    |   movel([0.327897, -1.235009, -2.660401, -0.816979, 1.570796, 1.898693],accel_mss,speed_ms,0,blend_radius_m)
    |   movel([0.327586, -1.234473, -2.660677, -0.817239, 1.570796, 1.898382],accel_mss,speed_ms,0,blend_radius_m)
    |   speed_ms = 0.005
    |   movel([0.327586, -1.224931, -2.656020, -0.831439, 1.570796, 1.898382],accel_mss,speed_ms,0,blend_radius_m)
    |   speed_ms = 0.040
    |   movel([0.337842, -1.232613, -2.652083, -0.827693, 1.570796, 1.908639],accel_mss,speed_ms,0,blend_radius_m)
    |   speed_ms = 0.005
    |   movel([0.337842, -1.242122, -2.656705, -0.813562, 1.570796, 1.908639],accel_mss,speed_ms,0,blend_radius_m)
    |   speed_ms = 0.025
    |   movel([0.336390, -1.242228, -2.656649, -0.813511, 1.570796, 1.907187],accel_mss,speed_ms,0,blend_radius_m)
    |   movel([0.335495, -1.242155, -2.656688, -0.813546, 1.570796, 1.906292],accel_mss,speed_ms,0,blend_radius_m)
    |   movel([0.333990, -1.241944, -2.656798, -0.813647, 1.570796, 1.904786],accel_mss,speed_ms,0,blend_radius_m)
    |   movel([0.333947, -1.242489, -2.656513, -0.813387, 1.570796, 1.904743],accel_mss,speed_ms,0,blend_radius_m)
    |   movel([0.333924, -1.243378, -2.656047, -0.812965, 1.570796, 1.904720],accel_mss,speed_ms,0,blend_radius_m)
    |   movel([0.333526, -1.244120, -2.655656, -0.812612, 1.570796, 1.904322],accel_mss,speed_ms,0,blend_radius_m)
    |   movel([0.333176, -1.244437, -2.655490, -0.812462, 1.570796, 1.903972],accel_mss,speed_ms,0,blend_radius_m)
    |   movel([0.332782, -1.244663, -2.655370, -0.812355, 1.570796, 1.903579],accel_mss,speed_ms,0,blend_radius_m)
    |   movel([0.331750, -1.244958, -2.655215, -0.812216, 1.570796, 1.902546],accel_mss,speed_ms,0,blend_radius_m)
    |   movel([0.330907, -1.245181, -2.655098, -0.812111, 1.570796, 1.901703],accel_mss,speed_ms,0,blend_radius_m)
    |   movel([0.331284, -1.245824, -2.654758, -0.811807, 1.570796, 1.902081],accel_mss,speed_ms,0,blend_radius_m)
    |   movel([0.331806, -1.246356, -2.654477, -0.811556, 1.570796, 1.902602],accel_mss,speed_ms,0,blend_radius_m)
    |   movel([0.333454, -1.247963, -2.653625, -0.810800, 1.570796, 1.904250],accel_mss,speed_ms,0,blend_radius_m)
    |   movel([0.333871, -1.248606, -2.653284, -0.810499, 1.570796, 1.904667],accel_mss,speed_ms,0,blend_radius_m)
    |   movel([0.333836, -1.249059, -2.653043, -0.810286, 1.570796, 1.904633],accel_mss,speed_ms,0,blend_radius_m)
    |   movel([0.333484, -1.249416, -2.652853, -0.810120, 1.570796, 1.904280],accel_mss,speed_ms,0,blend_radius_m)
    |   movel([0.333131, -1.249421, -2.652851, -0.810117, 1.570796, 1.903927],accel_mss,speed_ms,0,blend_radius_m)
    |   movel([0.332061, -1.248584, -2.653296, -0.810509, 1.570796, 1.902858],accel_mss,speed_ms,0,blend_radius_m)
    |   movel([0.329590, -1.246252, -2.654532, -0.811605, 1.570796, 1.900386],accel_mss,speed_ms,0,blend_radius_m)
    |   movel([0.329051, -1.245580, -2.654887, -0.811922, 1.570796, 1.899848],accel_mss,speed_ms,0,blend_radius_m)
    |   movel([0.328887, -1.245037, -2.655174, -0.812179, 1.570796, 1.899684],accel_mss,speed_ms,0,blend_radius_m)
    |   movel([0.329075, -1.244647, -2.655379, -0.812363, 1.570796, 1.899871],accel_mss,speed_ms,0,blend_radius_m)
    |   movel([0.329758, -1.244331, -2.655545, -0.812513, 1.570796, 1.900555],accel_mss,speed_ms,0,blend_radius_m)
    |   movel([0.330219, -1.244220, -2.655604, -0.812565, 1.570796, 1.901015],accel_mss,speed_ms,0,blend_radius_m)
    |   movel([0.332711, -1.243637, -2.655910, -0.812842, 1.570796, 1.903507],accel_mss,speed_ms,0,blend_radius_m)
    |   movel([0.332571, -1.242862, -2.656318, -0.813210, 1.570796, 1.903368],accel_mss,speed_ms,0,blend_radius_m)
    |   movel([0.332085, -1.240846, -2.657373, -0.814171, 1.570796, 1.902881],accel_mss,speed_ms,0,blend_radius_m)
    |   movel([0.332184, -1.240399, -2.657606, -0.814384, 1.570796, 1.902980],accel_mss,speed_ms,0,blend_radius_m)
    |   movel([0.332457, -1.240129, -2.657746, -0.814513, 1.570796, 1.903254],accel_mss,speed_ms,0,blend_radius_m)
    |   movel([0.332852, -1.240044, -2.657791, -0.814554, 1.570796, 1.903648],accel_mss,speed_ms,0,blend_radius_m)
    |   movel([0.335457, -1.240841, -2.657375, -0.814173, 1.570796, 1.906254],accel_mss,speed_ms,0,blend_radius_m)
    |   movel([0.336114, -1.240976, -2.657305, -0.814108, 1.570796, 1.906911],accel_mss,speed_ms,0,blend_radius_m)
    |   movel([0.337508, -1.240998, -2.657293, -0.814098, 1.570796, 1.908304],accel_mss,speed_ms,0,blend_radius_m)
    |   movel([0.338667, -1.240917, -2.657336, -0.814137, 1.570796, 1.909464],accel_mss,speed_ms,0,blend_radius_m)
    |   movel([0.339093, -1.240957, -2.657315, -0.814118, 1.570796, 1.909889],accel_mss,speed_ms,0,blend_radius_m)
    |   movel([0.339216, -1.241123, -2.657228, -0.814038, 1.570796, 1.910012],accel_mss,speed_ms,0,blend_radius_m)
    |   movel([0.338972, -1.241703, -2.656925, -0.813761, 1.570796, 1.909768],accel_mss,speed_ms,0,blend_radius_m)
    |   movel([0.338768, -1.241870, -2.656837, -0.813682, 1.570796, 1.909564],accel_mss,speed_ms,0,blend_radius_m)
    |   movel([0.337842, -1.242122, -2.656705, -0.813562, 1.570796, 1.908639],accel_mss,speed_ms,0,blend_radius_m)
    |   movel([0.336390, -1.242228, -2.656649, -0.813511, 1.570796, 1.907187],accel_mss,speed_ms,0,blend_radius_m)
    |   movel([0.335495, -1.242155, -2.656688, -0.813546, 1.570796, 1.906292],accel_mss,speed_ms,0,blend_radius_m)
    |   movel([0.335218, -1.242116, -2.656708, -0.813564, 1.570796, 1.906015],accel_mss,speed_ms,0,blend_radius_m)
    |   speed_ms = 0.005
    |   movel([0.335218, -1.232607, -2.652086, -0.827696, 1.570796, 1.906015],accel_mss,speed_ms,0,blend_radius_m)
    |   speed_ms = 0.040
    |   movel([0.344776, -1.237105, -2.649749, -0.825535, 1.570796, 1.915573],accel_mss,speed_ms,0,blend_radius_m)
    |   speed_ms = 0.005
    |   movel([0.344776, -1.246594, -2.654351, -0.811444, 1.570796, 1.915573],accel_mss,speed_ms,0,blend_radius_m)
    |   speed_ms = 0.025
    |   movel([0.344962, -1.247047, -2.654111, -0.811231, 1.570796, 1.915759],accel_mss,speed_ms,0,blend_radius_m)
    |   movel([0.345103, -1.247442, -2.653902, -0.811045, 1.570796, 1.915899],accel_mss,speed_ms,0,blend_radius_m)
    |   movel([0.345193, -1.247835, -2.653693, -0.810860, 1.570796, 1.915990],accel_mss,speed_ms,0,blend_radius_m)
    |   movel([0.343853, -1.247462, -2.653891, -0.811035, 1.570796, 1.914649],accel_mss,speed_ms,0,blend_radius_m)
    |   movel([0.343381, -1.247399, -2.653925, -0.811065, 1.570796, 1.914177],accel_mss,speed_ms,0,blend_radius_m)
    |   movel([0.342236, -1.247467, -2.653889, -0.811033, 1.570796, 1.913033],accel_mss,speed_ms,0,blend_radius_m)
    |   movel([0.340990, -1.247651, -2.653791, -0.810947, 1.570796, 1.911786],accel_mss,speed_ms,0,blend_radius_m)
    |   movel([0.341964, -1.245315, -2.655027, -0.812047, 1.570796, 1.912761],accel_mss,speed_ms,0,blend_radius_m)
    |   movel([0.342301, -1.244772, -2.655313, -0.812304, 1.570796, 1.913097],accel_mss,speed_ms,0,blend_radius_m)
    |   movel([0.342917, -1.244066, -2.655685, -0.812638, 1.570796, 1.913714],accel_mss,speed_ms,0,blend_radius_m)
    |   movel([0.343093, -1.244020, -2.655709, -0.812660, 1.570796, 1.913889],accel_mss,speed_ms,0,blend_radius_m)
    |   movel([0.343277, -1.244144, -2.655644, -0.812601, 1.570796, 1.914074],accel_mss,speed_ms,0,blend_radius_m)
    |   movel([0.343671, -1.244629, -2.655388, -0.812371, 1.570796, 1.914468],accel_mss,speed_ms,0,blend_radius_m)
    |   movel([0.344776, -1.246594, -2.654351, -0.811444, 1.570796, 1.915573],accel_mss,speed_ms,0,blend_radius_m)
    |   movel([0.344962, -1.247047, -2.654111, -0.811231, 1.570796, 1.915759],accel_mss,speed_ms,0,blend_radius_m)
    |   movel([0.345103, -1.247442, -2.653902, -0.811045, 1.570796, 1.915899],accel_mss,speed_ms,0,blend_radius_m)
    |   movel([0.345193, -1.247835, -2.653693, -0.810860, 1.570796, 1.915990],accel_mss,speed_ms,0,blend_radius_m)
    |   movel([0.344251, -1.247571, -2.653834, -0.810985, 1.570796, 1.915047],accel_mss,speed_ms,0,blend_radius_m)
    |   speed_ms = 0.005
    |   movel([0.344251, -1.238086, -2.649236, -0.825066, 1.570796, 1.915047],accel_mss,speed_ms,0,blend_radius_m)
    |   speed_ms = 0.040
    |   movel([0.347433, -1.243638, -2.646313, -0.822438, 1.570796, 1.918229],accel_mss,speed_ms,0,blend_radius_m)
    |   speed_ms = 0.005
    |   movel([0.347433, -1.253097, -2.650885, -0.808407, 1.570796, 1.918229],accel_mss,speed_ms,0,blend_radius_m)
    |   speed_ms = 0.025
    |   movel([0.347850, -1.253561, -2.650636, -0.808192, 1.570796, 1.918646],accel_mss,speed_ms,0,blend_radius_m)
    |   movel([0.346822, -1.254725, -2.650010, -0.807654, 1.570796, 1.917619],accel_mss,speed_ms,0,blend_radius_m)
    |   movel([0.346418, -1.255196, -2.649756, -0.807437, 1.570796, 1.917215],accel_mss,speed_ms,0,blend_radius_m)
    |   movel([0.345672, -1.256232, -2.649197, -0.806961, 1.570796, 1.916468],accel_mss,speed_ms,0,blend_radius_m)
    |   movel([0.345493, -1.256601, -2.648997, -0.806791, 1.570796, 1.916289],accel_mss,speed_ms,0,blend_radius_m)
    |   movel([0.345323, -1.256697, -2.648945, -0.806747, 1.570796, 1.916119],accel_mss,speed_ms,0,blend_radius_m)
    |   movel([0.345210, -1.256550, -2.649025, -0.806815, 1.570796, 1.916007],accel_mss,speed_ms,0,blend_radius_m)
    |   movel([0.345305, -1.255281, -2.649710, -0.807398, 1.570796, 1.916101],accel_mss,speed_ms,0,blend_radius_m)
    |   movel([0.345190, -1.254371, -2.650200, -0.807817, 1.570796, 1.915986],accel_mss,speed_ms,0,blend_radius_m)
    |   movel([0.344521, -1.252694, -2.651102, -0.808594, 1.570796, 1.915318],accel_mss,speed_ms,0,blend_radius_m)
    |   movel([0.343954, -1.251814, -2.651573, -0.809002, 1.570796, 1.914750],accel_mss,speed_ms,0,blend_radius_m)
    |   movel([0.345412, -1.251976, -2.651486, -0.808926, 1.570796, 1.916209],accel_mss,speed_ms,0,blend_radius_m)
    |   movel([0.346198, -1.252267, -2.651330, -0.808791, 1.570796, 1.916994],accel_mss,speed_ms,0,blend_radius_m)
    |   movel([0.347433, -1.253097, -2.650885, -0.808407, 1.570796, 1.918229],accel_mss,speed_ms,0,blend_radius_m)
    |   movel([0.347850, -1.253561, -2.650636, -0.808192, 1.570796, 1.918646],accel_mss,speed_ms,0,blend_radius_m)
    |   movel([0.346822, -1.254725, -2.650010, -0.807654, 1.570796, 1.917619],accel_mss,speed_ms,0,blend_radius_m)
    |   movel([0.346418, -1.255196, -2.649756, -0.807437, 1.570796, 1.917215],accel_mss,speed_ms,0,blend_radius_m)
    |   movel([0.346284, -1.255382, -2.649655, -0.807351, 1.570796, 1.917080],accel_mss,speed_ms,0,blend_radius_m)
    |   speed_ms = 0.005
    |   movel([0.346284, -1.245935, -2.645093, -0.821361, 1.570796, 1.917080],accel_mss,speed_ms,0,blend_radius_m)
    |   speed_ms = 0.040
    |   movel([0.344061, -1.246376, -2.644858, -0.821155, 1.570796, 1.914858],accel_mss,speed_ms,0,blend_radius_m)
    |   speed_ms = 0.005
    |   movel([0.344061, -1.255822, -2.649418, -0.807149, 1.570796, 1.914858],accel_mss,speed_ms,0,blend_radius_m)
    |   speed_ms = 0.025
    |   movel([0.344055, -1.256519, -2.649041, -0.806829, 1.570796, 1.914852],accel_mss,speed_ms,0,blend_radius_m)
    |   movel([0.343811, -1.256521, -2.649040, -0.806828, 1.570796, 1.914607],accel_mss,speed_ms,0,blend_radius_m)
    |   movel([0.343651, -1.256550, -2.649025, -0.806815, 1.570796, 1.914448],accel_mss,speed_ms,0,blend_radius_m)
    |   movel([0.342482, -1.257406, -2.648561, -0.806422, 1.570796, 1.913278],accel_mss,speed_ms,0,blend_radius_m)
    |   movel([0.341957, -1.257846, -2.648322, -0.806221, 1.570796, 1.912753],accel_mss,speed_ms,0,blend_radius_m)
    |   movel([0.338805, -1.260237, -2.647021, -0.805131, 1.570796, 1.909602],accel_mss,speed_ms,0,blend_radius_m)
    |   movel([0.338410, -1.260591, -2.646828, -0.804970, 1.570796, 1.909206],accel_mss,speed_ms,0,blend_radius_m)
    |   movel([0.338279, -1.260944, -2.646635, -0.804809, 1.570796, 1.909075],accel_mss,speed_ms,0,blend_radius_m)
    |   movel([0.338423, -1.261159, -2.646518, -0.804712, 1.570796, 1.909219],accel_mss,speed_ms,0,blend_radius_m)
    |   movel([0.339527, -1.261944, -2.646088, -0.804356, 1.570796, 1.910324],accel_mss,speed_ms,0,blend_radius_m)
    |   movel([0.339657, -1.262109, -2.645998, -0.804282, 1.570796, 1.910454],accel_mss,speed_ms,0,blend_radius_m)
    |   movel([0.339616, -1.262279, -2.645905, -0.804205, 1.570796, 1.910412],accel_mss,speed_ms,0,blend_radius_m)
    |   movel([0.339373, -1.262541, -2.645761, -0.804087, 1.570796, 1.910169],accel_mss,speed_ms,0,blend_radius_m)
    |   movel([0.336435, -1.264693, -2.644579, -0.803117, 1.570796, 1.907232],accel_mss,speed_ms,0,blend_radius_m)
    |   movel([0.335844, -1.265143, -2.644330, -0.802915, 1.570796, 1.906640],accel_mss,speed_ms,0,blend_radius_m)
    |   movel([0.335265, -1.265665, -2.644043, -0.802682, 1.570796, 1.906061],accel_mss,speed_ms,0,blend_radius_m)
    |   movel([0.335504, -1.266428, -2.643621, -0.802340, 1.570796, 1.906300],accel_mss,speed_ms,0,blend_radius_m)
    |   movel([0.335563, -1.266696, -2.643473, -0.802221, 1.570796, 1.906360],accel_mss,speed_ms,0,blend_radius_m)
    |   movel([0.335537, -1.267980, -2.642761, -0.801648, 1.570796, 1.906333],accel_mss,speed_ms,0,blend_radius_m)
    |   movel([0.332951, -1.269710, -2.641799, -0.800880, 1.570796, 1.903747],accel_mss,speed_ms,0,blend_radius_m)
    |   movel([0.330029, -1.271596, -2.640746, -0.800047, 1.570796, 1.900825],accel_mss,speed_ms,0,blend_radius_m)
    |   movel([0.329751, -1.271577, -2.640757, -0.800055, 1.570796, 1.900547],accel_mss,speed_ms,0,blend_radius_m)
    |   movel([0.329384, -1.270609, -2.641297, -0.800482, 1.570796, 1.900181],accel_mss,speed_ms,0,blend_radius_m)
    |   movel([0.329403, -1.269974, -2.641652, -0.800763, 1.570796, 1.900199],accel_mss,speed_ms,0,blend_radius_m)
    |   movel([0.329571, -1.269468, -2.641934, -0.800987, 1.570796, 1.900367],accel_mss,speed_ms,0,blend_radius_m)
    |   movel([0.329743, -1.269337, -2.642007, -0.801045, 1.570796, 1.900539],accel_mss,speed_ms,0,blend_radius_m)
    |   movel([0.331850, -1.268374, -2.642542, -0.801473, 1.570796, 1.902646],accel_mss,speed_ms,0,blend_radius_m)
    |   movel([0.333029, -1.267761, -2.642882, -0.801745, 1.570796, 1.903825],accel_mss,speed_ms,0,blend_radius_m)
    |   movel([0.333747, -1.265589, -2.644084, -0.802716, 1.570796, 1.904543],accel_mss,speed_ms,0,blend_radius_m)
    |   movel([0.334469, -1.263406, -2.645286, -0.803696, 1.570796, 1.905265],accel_mss,speed_ms,0,blend_radius_m)
    |   movel([0.336265, -1.262881, -2.645575, -0.803933, 1.570796, 1.907061],accel_mss,speed_ms,0,blend_radius_m)
    |   movel([0.336592, -1.262741, -2.645652, -0.803996, 1.570796, 1.907389],accel_mss,speed_ms,0,blend_radius_m)
    |   movel([0.336933, -1.262413, -2.645831, -0.804144, 1.570796, 1.907730],accel_mss,speed_ms,0,blend_radius_m)
    |   movel([0.337189, -1.261814, -2.646160, -0.804415, 1.570796, 1.907986],accel_mss,speed_ms,0,blend_radius_m)
    |   movel([0.338579, -1.257841, -2.648325, -0.806223, 1.570796, 1.909375],accel_mss,speed_ms,0,blend_radius_m)
    |   movel([0.339139, -1.256788, -2.648896, -0.806705, 1.570796, 1.909935],accel_mss,speed_ms,0,blend_radius_m)
    |   movel([0.339420, -1.256465, -2.649070, -0.806853, 1.570796, 1.910216],accel_mss,speed_ms,0,blend_radius_m)
    |   movel([0.339765, -1.256214, -2.649206, -0.806969, 1.570796, 1.910561],accel_mss,speed_ms,0,blend_radius_m)
    |   movel([0.340589, -1.255920, -2.649365, -0.807104, 1.570796, 1.911385],accel_mss,speed_ms,0,blend_radius_m)
    |   movel([0.341049, -1.255767, -2.649448, -0.807174, 1.570796, 1.911846],accel_mss,speed_ms,0,blend_radius_m)
    |   movel([0.341344, -1.255487, -2.649599, -0.807303, 1.570796, 1.912141],accel_mss,speed_ms,0,blend_radius_m)
    |   movel([0.341539, -1.254979, -2.649873, -0.807537, 1.570796, 1.912335],accel_mss,speed_ms,0,blend_radius_m)
    |   movel([0.341939, -1.252528, -2.651191, -0.808670, 1.570796, 1.912735],accel_mss,speed_ms,0,blend_radius_m)
    |   movel([0.342088, -1.252418, -2.651250, -0.808722, 1.570796, 1.912884],accel_mss,speed_ms,0,blend_radius_m)
    |   movel([0.342330, -1.252471, -2.651221, -0.808697, 1.570796, 1.913126],accel_mss,speed_ms,0,blend_radius_m)
    |   movel([0.343006, -1.252992, -2.650942, -0.808455, 1.570796, 1.913803],accel_mss,speed_ms,0,blend_radius_m)
    |   movel([0.343564, -1.253810, -2.650502, -0.808077, 1.570796, 1.914360],accel_mss,speed_ms,0,blend_radius_m)
    |   movel([0.343936, -1.254798, -2.649970, -0.807621, 1.570796, 1.914733],accel_mss,speed_ms,0,blend_radius_m)
    |   movel([0.344061, -1.255822, -2.649418, -0.807149, 1.570796, 1.914858],accel_mss,speed_ms,0,blend_radius_m)
    |   movel([0.344055, -1.256519, -2.649041, -0.806829, 1.570796, 1.914852],accel_mss,speed_ms,0,blend_radius_m)
    |   movel([0.343811, -1.256521, -2.649040, -0.806828, 1.570796, 1.914607],accel_mss,speed_ms,0,blend_radius_m)
    |   movel([0.343651, -1.256550, -2.649025, -0.806815, 1.570796, 1.914448],accel_mss,speed_ms,0,blend_radius_m)
    |   movel([0.342482, -1.257406, -2.648561, -0.806422, 1.570796, 1.913278],accel_mss,speed_ms,0,blend_radius_m)
    |   movel([0.342098, -1.257728, -2.648386, -0.806275, 1.570796, 1.912895],accel_mss,speed_ms,0,blend_radius_m)
    |   speed_ms = 0.005
    |   movel([0.342098, -1.248291, -2.643835, -0.820263, 1.570796, 1.912895],accel_mss,speed_ms,0,blend_radius_m)
    |   speed_ms = 0.040
    |   movel([0.340847, -1.242148, -2.647101, -0.823140, 1.570796, 1.911643],accel_mss,speed_ms,0,blend_radius_m)
    |   speed_ms = 0.005
    |   movel([0.340847, -1.251613, -2.651681, -0.809095, 1.570796, 1.911643],accel_mss,speed_ms,0,blend_radius_m)
    |   speed_ms = 0.025
    |   movel([0.341030, -1.249021, -2.653063, -0.810304, 1.570796, 1.911826],accel_mss,speed_ms,0,blend_radius_m)
    |   movel([0.340905, -1.248934, -2.653110, -0.810345, 1.570796, 1.911701],accel_mss,speed_ms,0,blend_radius_m)
    |   movel([0.340717, -1.249064, -2.653041, -0.810285, 1.570796, 1.911513],accel_mss,speed_ms,0,blend_radius_m)
    |   movel([0.340472, -1.249484, -2.652817, -0.810088, 1.570796, 1.911268],accel_mss,speed_ms,0,blend_radius_m)
    |   movel([0.337881, -1.255319, -2.649690, -0.807381, 1.570796, 1.908678],accel_mss,speed_ms,0,blend_radius_m)
    |   movel([0.336934, -1.257061, -2.648748, -0.806580, 1.570796, 1.907730],accel_mss,speed_ms,0,blend_radius_m)
    |   movel([0.334763, -1.260390, -2.646938, -0.805061, 1.570796, 1.905559],accel_mss,speed_ms,0,blend_radius_m)
    |   movel([0.333555, -1.261957, -2.646081, -0.804351, 1.570796, 1.904351],accel_mss,speed_ms,0,blend_radius_m)
    |   movel([0.330890, -1.264905, -2.644462, -0.803022, 1.570796, 1.901686],accel_mss,speed_ms,0,blend_radius_m)
    |   movel([0.329911, -1.265954, -2.643883, -0.802552, 1.570796, 1.900707],accel_mss,speed_ms,0,blend_radius_m)
    |   movel([0.329256, -1.266827, -2.643400, -0.802162, 1.570796, 1.900052],accel_mss,speed_ms,0,blend_radius_m)
    |   movel([0.328578, -1.268019, -2.642739, -0.801631, 1.570796, 1.899374],accel_mss,speed_ms,0,blend_radius_m)
    |   movel([0.325671, -1.273695, -2.639569, -0.799125, 1.570796, 1.896467],accel_mss,speed_ms,0,blend_radius_m)
    |   movel([0.325528, -1.273943, -2.639430, -0.799016, 1.570796, 1.896324],accel_mss,speed_ms,0,blend_radius_m)
    |   movel([0.325367, -1.274331, -2.639211, -0.798846, 1.570796, 1.896164],accel_mss,speed_ms,0,blend_radius_m)
    |   movel([0.328357, -1.272726, -2.640113, -0.799550, 1.570796, 1.899153],accel_mss,speed_ms,0,blend_radius_m)
    |   movel([0.328194, -1.270494, -2.641362, -0.800533, 1.570796, 1.898990],accel_mss,speed_ms,0,blend_radius_m)
    |   movel([0.328220, -1.269995, -2.641640, -0.800754, 1.570796, 1.899016],accel_mss,speed_ms,0,blend_radius_m)
    |   movel([0.328503, -1.268871, -2.642266, -0.801252, 1.570796, 1.899299],accel_mss,speed_ms,0,blend_radius_m)
    |   movel([0.329810, -1.268303, -2.642582, -0.801504, 1.570796, 1.900606],accel_mss,speed_ms,0,blend_radius_m)
    |   movel([0.331265, -1.267638, -2.642951, -0.801800, 1.570796, 1.902062],accel_mss,speed_ms,0,blend_radius_m)
    |   movel([0.331801, -1.267237, -2.643173, -0.801979, 1.570796, 1.902597],accel_mss,speed_ms,0,blend_radius_m)
    |   movel([0.332158, -1.266675, -2.643484, -0.802230, 1.570796, 1.902955],accel_mss,speed_ms,0,blend_radius_m)
    |   movel([0.332753, -1.265078, -2.644366, -0.802945, 1.570796, 1.903549],accel_mss,speed_ms,0,blend_radius_m)
    |   movel([0.333371, -1.263441, -2.645267, -0.803681, 1.570796, 1.904167],accel_mss,speed_ms,0,blend_radius_m)
    |   movel([0.333801, -1.262717, -2.645665, -0.804007, 1.570796, 1.904597],accel_mss,speed_ms,0,blend_radius_m)
    |   movel([0.334329, -1.262314, -2.645886, -0.804189, 1.570796, 1.905125],accel_mss,speed_ms,0,blend_radius_m)
    |   movel([0.335176, -1.262051, -2.646030, -0.804308, 1.570796, 1.905973],accel_mss,speed_ms,0,blend_radius_m)
    |   movel([0.336100, -1.261871, -2.646128, -0.804390, 1.570796, 1.906896],accel_mss,speed_ms,0,blend_radius_m)
    |   movel([0.336424, -1.260706, -2.646766, -0.804918, 1.570796, 1.907221],accel_mss,speed_ms,0,blend_radius_m)
    |   movel([0.337089, -1.258609, -2.647908, -0.805872, 1.570796, 1.907885],accel_mss,speed_ms,0,blend_radius_m)
    |   movel([0.337773, -1.257133, -2.648709, -0.806547, 1.570796, 1.908570],accel_mss,speed_ms,0,blend_radius_m)
    |   movel([0.338562, -1.256069, -2.649284, -0.807036, 1.570796, 1.909358],accel_mss,speed_ms,0,blend_radius_m)
    |   movel([0.339534, -1.255278, -2.649712, -0.807399, 1.570796, 1.910330],accel_mss,speed_ms,0,blend_radius_m)
    |   movel([0.340367, -1.254662, -2.650044, -0.807684, 1.570796, 1.911163],accel_mss,speed_ms,0,blend_radius_m)
    |   movel([0.340847, -1.251613, -2.651681, -0.809095, 1.570796, 1.911643],accel_mss,speed_ms,0,blend_radius_m)
    |   movel([0.341030, -1.249021, -2.653063, -0.810304, 1.570796, 1.911826],accel_mss,speed_ms,0,blend_radius_m)
    |   speed_ms = 0.005
    |   movel([0.341030, -1.239544, -2.648472, -0.824373, 1.570796, 1.911826],accel_mss,speed_ms,0,blend_radius_m)
    |   speed_ms = 0.040
    |   movel([0.331737, -1.240212, -2.648121, -0.824056, 1.570796, 1.902534],accel_mss,speed_ms,0,blend_radius_m)
    |   speed_ms = 0.005
    |   movel([0.331737, -1.249686, -2.652709, -0.809993, 1.570796, 1.902534],accel_mss,speed_ms,0,blend_radius_m)
    |   speed_ms = 0.025
    |   movel([0.330795, -1.250056, -2.652512, -0.809821, 1.570796, 1.901591],accel_mss,speed_ms,0,blend_radius_m)
    |   movel([0.329929, -1.250332, -2.652365, -0.809692, 1.570796, 1.900726],accel_mss,speed_ms,0,blend_radius_m)
    |   movel([0.326537, -1.251391, -2.651800, -0.809199, 1.570796, 1.897333],accel_mss,speed_ms,0,blend_radius_m)
    |   movel([0.326526, -1.251596, -2.651690, -0.809103, 1.570796, 1.897322],accel_mss,speed_ms,0,blend_radius_m)
    |   movel([0.327723, -1.251755, -2.651605, -0.809029, 1.570796, 1.898519],accel_mss,speed_ms,0,blend_radius_m)
    |   movel([0.329778, -1.251841, -2.651558, -0.808989, 1.570796, 1.900574],accel_mss,speed_ms,0,blend_radius_m)
    |   movel([0.329907, -1.251902, -2.651526, -0.808961, 1.570796, 1.900703],accel_mss,speed_ms,0,blend_radius_m)
    |   movel([0.329913, -1.252302, -2.651312, -0.808775, 1.570796, 1.900710],accel_mss,speed_ms,0,blend_radius_m)
    |   movel([0.329809, -1.252608, -2.651148, -0.808633, 1.570796, 1.900605],accel_mss,speed_ms,0,blend_radius_m)
    |   movel([0.329652, -1.252785, -2.651053, -0.808551, 1.570796, 1.900448],accel_mss,speed_ms,0,blend_radius_m)
    |   movel([0.329377, -1.252917, -2.650982, -0.808490, 1.570796, 1.900174],accel_mss,speed_ms,0,blend_radius_m)
    |   movel([0.327349, -1.253469, -2.650685, -0.808234, 1.570796, 1.898145],accel_mss,speed_ms,0,blend_radius_m)
    |   movel([0.327069, -1.253650, -2.650588, -0.808151, 1.570796, 1.897865],accel_mss,speed_ms,0,blend_radius_m)
    |   movel([0.327040, -1.253845, -2.650484, -0.808061, 1.570796, 1.897836],accel_mss,speed_ms,0,blend_radius_m)
    |   movel([0.327661, -1.254243, -2.650269, -0.807877, 1.570796, 1.898457],accel_mss,speed_ms,0,blend_radius_m)
    |   movel([0.328324, -1.254731, -2.650006, -0.807651, 1.570796, 1.899120],accel_mss,speed_ms,0,blend_radius_m)
    |   movel([0.328392, -1.255160, -2.649775, -0.807454, 1.570796, 1.899188],accel_mss,speed_ms,0,blend_radius_m)
    |   movel([0.328033, -1.255565, -2.649557, -0.807267, 1.570796, 1.898830],accel_mss,speed_ms,0,blend_radius_m)
    |   movel([0.327106, -1.255967, -2.649340, -0.807082, 1.570796, 1.897902],accel_mss,speed_ms,0,blend_radius_m)
    |   movel([0.323428, -1.257420, -2.648553, -0.806416, 1.570796, 1.894225],accel_mss,speed_ms,0,blend_radius_m)
    |   movel([0.324422, -1.257532, -2.648492, -0.806364, 1.570796, 1.895219],accel_mss,speed_ms,0,blend_radius_m)
    |   movel([0.327337, -1.258004, -2.648236, -0.806149, 1.570796, 1.898134],accel_mss,speed_ms,0,blend_radius_m)
    |   movel([0.328343, -1.258263, -2.648096, -0.806030, 1.570796, 1.899139],accel_mss,speed_ms,0,blend_radius_m)
    |   movel([0.328504, -1.258474, -2.647981, -0.805934, 1.570796, 1.899301],accel_mss,speed_ms,0,blend_radius_m)
    |   movel([0.328399, -1.258767, -2.647822, -0.805800, 1.570796, 1.899196],accel_mss,speed_ms,0,blend_radius_m)
    |   movel([0.328100, -1.259069, -2.647658, -0.805662, 1.570796, 1.898897],accel_mss,speed_ms,0,blend_radius_m)
    |   movel([0.327511, -1.259438, -2.647457, -0.805494, 1.570796, 1.898308],accel_mss,speed_ms,0,blend_radius_m)
    |   movel([0.324829, -1.260884, -2.646668, -0.804837, 1.570796, 1.895626],accel_mss,speed_ms,0,blend_radius_m)
    |   movel([0.322733, -1.262208, -2.645944, -0.804237, 1.570796, 1.893529],accel_mss,speed_ms,0,blend_radius_m)
    |   movel([0.318382, -1.265269, -2.644261, -0.802859, 1.570796, 1.889179],accel_mss,speed_ms,0,blend_radius_m)
    |   movel([0.317603, -1.265850, -2.643940, -0.802599, 1.570796, 1.888400],accel_mss,speed_ms,0,blend_radius_m)
    |   movel([0.316328, -1.266748, -2.643444, -0.802197, 1.570796, 1.887124],accel_mss,speed_ms,0,blend_radius_m)
    |   movel([0.316171, -1.266813, -2.643408, -0.802168, 1.570796, 1.886967],accel_mss,speed_ms,0,blend_radius_m)
    |   movel([0.315790, -1.266570, -2.643543, -0.802277, 1.570796, 1.886587],accel_mss,speed_ms,0,blend_radius_m)
    |   movel([0.315751, -1.266387, -2.643644, -0.802359, 1.570796, 1.886548],accel_mss,speed_ms,0,blend_radius_m)
    |   movel([0.316070, -1.265956, -2.643882, -0.802551, 1.570796, 1.886867],accel_mss,speed_ms,0,blend_radius_m)
    |   movel([0.316633, -1.265500, -2.644134, -0.802756, 1.570796, 1.887429],accel_mss,speed_ms,0,blend_radius_m)
    |   movel([0.320336, -1.262735, -2.645655, -0.803999, 1.570796, 1.891132],accel_mss,speed_ms,0,blend_radius_m)
    |   movel([0.322202, -1.261450, -2.646359, -0.804580, 1.570796, 1.892998],accel_mss,speed_ms,0,blend_radius_m)
    |   movel([0.325319, -1.259432, -2.647460, -0.805497, 1.570796, 1.896115],accel_mss,speed_ms,0,blend_radius_m)
    |   movel([0.325768, -1.259095, -2.647644, -0.805650, 1.570796, 1.896564],accel_mss,speed_ms,0,blend_radius_m)
    |   movel([0.325072, -1.258883, -2.647759, -0.805747, 1.570796, 1.895868],accel_mss,speed_ms,0,blend_radius_m)
    |   movel([0.320430, -1.258455, -2.647992, -0.805943, 1.570796, 1.891226],accel_mss,speed_ms,0,blend_radius_m)
    |   movel([0.320318, -1.258395, -2.648024, -0.805970, 1.570796, 1.891115],accel_mss,speed_ms,0,blend_radius_m)
    |   movel([0.320419, -1.258013, -2.648231, -0.806144, 1.570796, 1.891215],accel_mss,speed_ms,0,blend_radius_m)
    |   movel([0.320535, -1.257847, -2.648322, -0.806220, 1.570796, 1.891331],accel_mss,speed_ms,0,blend_radius_m)
    |   movel([0.320815, -1.257606, -2.648453, -0.806331, 1.570796, 1.891611],accel_mss,speed_ms,0,blend_radius_m)
    |   movel([0.321422, -1.257271, -2.648634, -0.806484, 1.570796, 1.892219],accel_mss,speed_ms,0,blend_radius_m)
    |   movel([0.326116, -1.255217, -2.649744, -0.807427, 1.570796, 1.896912],accel_mss,speed_ms,0,blend_radius_m)
    |   movel([0.325392, -1.254648, -2.650051, -0.807690, 1.570796, 1.896189],accel_mss,speed_ms,0,blend_radius_m)
    |   movel([0.324878, -1.254251, -2.650265, -0.807873, 1.570796, 1.895675],accel_mss,speed_ms,0,blend_radius_m)
    |   movel([0.324731, -1.253850, -2.650481, -0.808058, 1.570796, 1.895527],accel_mss,speed_ms,0,blend_radius_m)
    |   movel([0.324926, -1.253489, -2.650675, -0.808225, 1.570796, 1.895723],accel_mss,speed_ms,0,blend_radius_m)
    |   movel([0.325765, -1.253000, -2.650937, -0.808451, 1.570796, 1.896562],accel_mss,speed_ms,0,blend_radius_m)
    |   movel([0.325811, -1.252840, -2.651023, -0.808526, 1.570796, 1.896608],accel_mss,speed_ms,0,blend_radius_m)
    |   movel([0.324383, -1.252610, -2.651147, -0.808632, 1.570796, 1.895179],accel_mss,speed_ms,0,blend_radius_m)
    |   movel([0.323248, -1.252478, -2.651218, -0.808694, 1.570796, 1.894045],accel_mss,speed_ms,0,blend_radius_m)
    |   movel([0.322708, -1.252302, -2.651312, -0.808775, 1.570796, 1.893504],accel_mss,speed_ms,0,blend_radius_m)
    |   movel([0.322573, -1.252042, -2.651451, -0.808896, 1.570796, 1.893369],accel_mss,speed_ms,0,blend_radius_m)
    |   movel([0.322732, -1.251685, -2.651642, -0.809062, 1.570796, 1.893528],accel_mss,speed_ms,0,blend_radius_m)
    |   movel([0.323093, -1.251363, -2.651814, -0.809212, 1.570796, 1.893889],accel_mss,speed_ms,0,blend_radius_m)
    |   movel([0.323501, -1.251161, -2.651922, -0.809305, 1.570796, 1.894297],accel_mss,speed_ms,0,blend_radius_m)
    |   movel([0.327531, -1.249933, -2.652578, -0.809878, 1.570796, 1.898327],accel_mss,speed_ms,0,blend_radius_m)
    |   movel([0.331601, -1.248763, -2.653201, -0.810425, 1.570796, 1.902397],accel_mss,speed_ms,0,blend_radius_m)
    |   movel([0.331890, -1.248761, -2.653202, -0.810426, 1.570796, 1.902686],accel_mss,speed_ms,0,blend_radius_m)
    |   movel([0.332103, -1.249173, -2.652983, -0.810233, 1.570796, 1.902900],accel_mss,speed_ms,0,blend_radius_m)
    |   movel([0.332078, -1.249339, -2.652894, -0.810156, 1.570796, 1.902874],accel_mss,speed_ms,0,blend_radius_m)
    |   movel([0.331737, -1.249686, -2.652709, -0.809993, 1.570796, 1.902534],accel_mss,speed_ms,0,blend_radius_m)
    |   movel([0.330795, -1.250056, -2.652512, -0.809821, 1.570796, 1.901591],accel_mss,speed_ms,0,blend_radius_m)
    |   movel([0.329929, -1.250332, -2.652365, -0.809692, 1.570796, 1.900726],accel_mss,speed_ms,0,blend_radius_m)
    |   movel([0.328825, -1.250676, -2.652182, -0.809531, 1.570796, 1.899621],accel_mss,speed_ms,0,blend_radius_m)
    |   speed_ms = 0.005
    |   movel([0.328825, -1.241206, -2.647598, -0.823585, 1.570796, 1.899621],accel_mss,speed_ms,0,blend_radius_m)
    |   speed_ms = 0.040
    |   movel([0.318480, -1.246370, -2.644861, -0.821158, 1.570796, 1.889276],accel_mss,speed_ms,0,blend_radius_m)
    |   speed_ms = 0.005
    |   movel([0.318480, -1.255816, -2.649421, -0.807152, 1.570796, 1.889276],accel_mss,speed_ms,0,blend_radius_m)
    |   speed_ms = 0.025
    |   movel([0.318409, -1.256197, -2.649215, -0.806977, 1.570796, 1.889205],accel_mss,speed_ms,0,blend_radius_m)
    |   movel([0.318480, -1.255816, -2.649421, -0.807152, 1.570796, 1.889276],accel_mss,speed_ms,0,blend_radius_m)
    |   movel([0.318409, -1.256197, -2.649215, -0.806977, 1.570796, 1.889205],accel_mss,speed_ms,0,blend_radius_m)
    |   movel([0.318480, -1.255816, -2.649421, -0.807152, 1.570796, 1.889276],accel_mss,speed_ms,0,blend_radius_m)
    |   speed_ms = 0.005
    |   movel([0.318480, -1.246370, -2.644861, -0.821158, 1.570796, 1.889276],accel_mss,speed_ms,0,blend_radius_m)
    |   speed_ms = 0.040
    |   movel([0.317236, -1.248446, -2.643752, -0.820191, 1.570796, 1.888032],accel_mss,speed_ms,0,blend_radius_m)
    |   speed_ms = 0.005
    |   movel([0.317236, -1.257881, -2.648303, -0.806205, 1.570796, 1.888032],accel_mss,speed_ms,0,blend_radius_m)
    |   speed_ms = 0.025
    |   movel([0.317126, -1.258257, -2.648099, -0.806033, 1.570796, 1.887922],accel_mss,speed_ms,0,blend_radius_m)
    |   movel([0.317353, -1.257837, -2.648327, -0.806225, 1.570796, 1.888149],accel_mss,speed_ms,0,blend_radius_m)
    |   movel([0.317126, -1.258257, -2.648099, -0.806033, 1.570796, 1.887922],accel_mss,speed_ms,0,blend_radius_m)
    |   movel([0.317353, -1.257837, -2.648327, -0.806225, 1.570796, 1.888149],accel_mss,speed_ms,0,blend_radius_m)
    |   speed_ms = 0.005
    |   movel([0.317353, -1.248401, -2.643776, -0.820212, 1.570796, 1.888149],accel_mss,speed_ms,0,blend_radius_m)
    |   speed_ms = 0.040
    |   movel([0.315637, -1.251072, -2.642342, -0.818975, 1.570796, 1.886433],accel_mss,speed_ms,0,blend_radius_m)
    |   speed_ms = 0.005
    |   movel([0.315637, -1.260495, -2.646881, -0.805013, 1.570796, 1.886433],accel_mss,speed_ms,0,blend_radius_m)
    |   speed_ms = 0.025
    |   movel([0.314421, -1.262568, -2.645747, -0.804075, 1.570796, 1.885218],accel_mss,speed_ms,0,blend_radius_m)
    |   movel([0.314110, -1.263358, -2.645313, -0.803718, 1.570796, 1.884907],accel_mss,speed_ms,0,blend_radius_m)
    |   movel([0.313273, -1.266414, -2.643629, -0.802347, 1.570796, 1.884070],accel_mss,speed_ms,0,blend_radius_m)
    |   movel([0.313132, -1.267147, -2.643223, -0.802019, 1.570796, 1.883929],accel_mss,speed_ms,0,blend_radius_m)
    |   movel([0.313157, -1.267750, -2.642889, -0.801751, 1.570796, 1.883953],accel_mss,speed_ms,0,blend_radius_m)
    |   movel([0.315232, -1.262096, -2.646005, -0.804288, 1.570796, 1.886029],accel_mss,speed_ms,0,blend_radius_m)
    |   movel([0.315671, -1.261056, -2.646574, -0.804759, 1.570796, 1.886467],accel_mss,speed_ms,0,blend_radius_m)
    |   movel([0.316908, -1.258688, -2.647865, -0.805836, 1.570796, 1.887704],accel_mss,speed_ms,0,blend_radius_m)
    |   movel([0.316718, -1.258811, -2.647798, -0.805780, 1.570796, 1.887514],accel_mss,speed_ms,0,blend_radius_m)
    |   movel([0.315637, -1.260495, -2.646881, -0.805013, 1.570796, 1.886433],accel_mss,speed_ms,0,blend_radius_m)
    |   movel([0.314421, -1.262568, -2.645747, -0.804075, 1.570796, 1.885218],accel_mss,speed_ms,0,blend_radius_m)
    |   movel([0.314154, -1.263247, -2.645374, -0.803768, 1.570796, 1.884951],accel_mss,speed_ms,0,blend_radius_m)
    |   speed_ms = 0.005
    |   movel([0.314154, -1.253838, -2.640847, -0.817704, 1.570796, 1.884951],accel_mss,speed_ms,0,blend_radius_m)
    |   speed_ms = 0.040
    |   movel([0.306668, -1.266775, -2.633735, -0.811879, 1.570796, 1.877464],accel_mss,speed_ms,0,blend_radius_m)
    |   speed_ms = 0.005
    |   movel([0.306668, -1.276119, -2.638203, -0.798067, 1.570796, 1.877464],accel_mss,speed_ms,0,blend_radius_m)
    |   speed_ms = 0.025
    |   movel([0.307047, -1.275960, -2.638293, -0.798136, 1.570796, 1.877844],accel_mss,speed_ms,0,blend_radius_m)
    |   movel([0.307298, -1.275670, -2.638457, -0.798262, 1.570796, 1.878095],accel_mss,speed_ms,0,blend_radius_m)
    |   movel([0.307403, -1.275216, -2.638713, -0.798460, 1.570796, 1.878200],accel_mss,speed_ms,0,blend_radius_m)
    |   movel([0.307351, -1.274575, -2.639074, -0.798740, 1.570796, 1.878148],accel_mss,speed_ms,0,blend_radius_m)
    |   movel([0.307088, -1.273570, -2.639639, -0.799180, 1.570796, 1.877884],accel_mss,speed_ms,0,blend_radius_m)
    |   movel([0.306641, -1.272687, -2.640135, -0.799567, 1.570796, 1.877438],accel_mss,speed_ms,0,blend_radius_m)
    |   movel([0.306021, -1.271952, -2.640547, -0.799890, 1.570796, 1.876818],accel_mss,speed_ms,0,blend_radius_m)
    |   movel([0.305235, -1.271377, -2.640869, -0.800143, 1.570796, 1.876031],accel_mss,speed_ms,0,blend_radius_m)
    |   movel([0.304299, -1.270974, -2.641094, -0.800321, 1.570796, 1.875096],accel_mss,speed_ms,0,blend_radius_m)
    |   movel([0.303237, -1.270753, -2.641217, -0.800419, 1.570796, 1.874033],accel_mss,speed_ms,0,blend_radius_m)
    |   movel([0.302056, -1.270716, -2.641238, -0.800435, 1.570796, 1.872852],accel_mss,speed_ms,0,blend_radius_m)
    |   movel([0.299811, -1.271036, -2.641059, -0.800294, 1.570796, 1.870607],accel_mss,speed_ms,0,blend_radius_m)
    |   movel([0.299436, -1.271046, -2.641054, -0.800289, 1.570796, 1.870233],accel_mss,speed_ms,0,blend_radius_m)
    |   movel([0.299084, -1.270646, -2.641277, -0.800466, 1.570796, 1.869880],accel_mss,speed_ms,0,blend_radius_m)
    |   movel([0.298752, -1.270045, -2.641612, -0.800732, 1.570796, 1.869548],accel_mss,speed_ms,0,blend_radius_m)
    |   movel([0.297298, -1.268697, -2.642363, -0.801329, 1.570796, 1.868094],accel_mss,speed_ms,0,blend_radius_m)
    |   movel([0.296564, -1.268302, -2.642582, -0.801505, 1.570796, 1.867360],accel_mss,speed_ms,0,blend_radius_m)
    |   movel([0.295674, -1.268094, -2.642698, -0.801597, 1.570796, 1.866470],accel_mss,speed_ms,0,blend_radius_m)
    |   movel([0.295213, -1.268125, -2.642681, -0.801584, 1.570796, 1.866009],accel_mss,speed_ms,0,blend_radius_m)
    |   movel([0.293435, -1.268519, -2.642462, -0.801408, 1.570796, 1.864231],accel_mss,speed_ms,0,blend_radius_m)
    |   movel([0.293929, -1.266685, -2.643479, -0.802225, 1.570796, 1.864726],accel_mss,speed_ms,0,blend_radius_m)
    |   movel([0.294456, -1.265010, -2.644404, -0.802975, 1.570796, 1.865252],accel_mss,speed_ms,0,blend_radius_m)
    |   movel([0.294715, -1.264562, -2.644651, -0.803176, 1.570796, 1.865511],accel_mss,speed_ms,0,blend_radius_m)
    |   movel([0.295801, -1.263380, -2.645301, -0.803708, 1.570796, 1.866597],accel_mss,speed_ms,0,blend_radius_m)
    |   movel([0.296555, -1.262857, -2.645588, -0.803944, 1.570796, 1.867351],accel_mss,speed_ms,0,blend_radius_m)
    |   movel([0.297392, -1.262483, -2.645793, -0.804113, 1.570796, 1.868189],accel_mss,speed_ms,0,blend_radius_m)
    |   movel([0.298326, -1.262248, -2.645922, -0.804219, 1.570796, 1.869122],accel_mss,speed_ms,0,blend_radius_m)
    |   movel([0.299194, -1.262188, -2.645955, -0.804246, 1.570796, 1.869991],accel_mss,speed_ms,0,blend_radius_m)
    |   movel([0.299864, -1.262327, -2.645878, -0.804183, 1.570796, 1.870660],accel_mss,speed_ms,0,blend_radius_m)
    |   movel([0.300504, -1.262725, -2.645660, -0.804003, 1.570796, 1.871301],accel_mss,speed_ms,0,blend_radius_m)
    |   movel([0.301309, -1.263508, -2.645231, -0.803651, 1.570796, 1.872105],accel_mss,speed_ms,0,blend_radius_m)
    |   movel([0.302639, -1.264630, -2.644613, -0.803146, 1.570796, 1.873436],accel_mss,speed_ms,0,blend_radius_m)
    |   movel([0.303331, -1.264856, -2.644489, -0.803044, 1.570796, 1.874128],accel_mss,speed_ms,0,blend_radius_m)
    |   movel([0.305497, -1.265267, -2.644262, -0.802860, 1.570796, 1.876293],accel_mss,speed_ms,0,blend_radius_m)
    |   movel([0.306236, -1.265740, -2.644001, -0.802648, 1.570796, 1.877033],accel_mss,speed_ms,0,blend_radius_m)
    |   movel([0.306724, -1.266521, -2.643569, -0.802298, 1.570796, 1.877521],accel_mss,speed_ms,0,blend_radius_m)
    |   movel([0.307042, -1.267718, -2.642907, -0.801765, 1.570796, 1.877838],accel_mss,speed_ms,0,blend_radius_m)
    |   movel([0.307338, -1.269622, -2.641848, -0.800919, 1.570796, 1.878134],accel_mss,speed_ms,0,blend_radius_m)
    |   movel([0.307443, -1.269708, -2.641800, -0.800881, 1.570796, 1.878239],accel_mss,speed_ms,0,blend_radius_m)
    |   movel([0.308131, -1.269671, -2.641821, -0.800897, 1.570796, 1.878927],accel_mss,speed_ms,0,blend_radius_m)
    |   movel([0.308275, -1.269576, -2.641873, -0.800939, 1.570796, 1.879072],accel_mss,speed_ms,0,blend_radius_m)
    |   movel([0.308418, -1.269054, -2.642164, -0.801171, 1.570796, 1.879214],accel_mss,speed_ms,0,blend_radius_m)
    |   movel([0.308420, -1.268135, -2.642675, -0.801579, 1.570796, 1.879216],accel_mss,speed_ms,0,blend_radius_m)
    |   movel([0.307841, -1.265652, -2.644050, -0.802688, 1.570796, 1.878637],accel_mss,speed_ms,0,blend_radius_m)
    |   movel([0.307463, -1.264949, -2.644437, -0.803002, 1.570796, 1.878260],accel_mss,speed_ms,0,blend_radius_m)
    |   movel([0.306557, -1.264173, -2.644865, -0.803351, 1.570796, 1.877354],accel_mss,speed_ms,0,blend_radius_m)
    |   movel([0.305989, -1.263989, -2.644966, -0.803434, 1.570796, 1.876785],accel_mss,speed_ms,0,blend_radius_m)
    |   movel([0.304271, -1.263725, -2.645111, -0.803553, 1.570796, 1.875067],accel_mss,speed_ms,0,blend_radius_m)
    |   movel([0.303525, -1.263453, -2.645261, -0.803675, 1.570796, 1.874321],accel_mss,speed_ms,0,blend_radius_m)
    |   movel([0.302066, -1.262284, -2.645902, -0.804203, 1.570796, 1.872863],accel_mss,speed_ms,0,blend_radius_m)
    |   movel([0.301186, -1.261515, -2.646323, -0.804551, 1.570796, 1.871983],accel_mss,speed_ms,0,blend_radius_m)
    |   movel([0.300359, -1.261116, -2.646542, -0.804732, 1.570796, 1.871155],accel_mss,speed_ms,0,blend_radius_m)
    |   movel([0.299424, -1.261018, -2.646595, -0.804776, 1.570796, 1.870220],accel_mss,speed_ms,0,blend_radius_m)
    |   movel([0.297548, -1.261365, -2.646405, -0.804619, 1.570796, 1.868345],accel_mss,speed_ms,0,blend_radius_m)
    |   movel([0.296995, -1.261565, -2.646296, -0.804528, 1.570796, 1.867792],accel_mss,speed_ms,0,blend_radius_m)
    |   movel([0.295947, -1.262154, -2.645973, -0.804261, 1.570796, 1.866743],accel_mss,speed_ms,0,blend_radius_m)
    |   movel([0.294969, -1.262822, -2.645607, -0.803960, 1.570796, 1.865765],accel_mss,speed_ms,0,blend_radius_m)
    |   movel([0.296415, -1.258144, -2.648161, -0.806085, 1.570796, 1.867211],accel_mss,speed_ms,0,blend_radius_m)
    |   movel([0.297876, -1.253426, -2.650709, -0.808254, 1.570796, 1.868673],accel_mss,speed_ms,0,blend_radius_m)
    |   movel([0.298521, -1.253192, -2.650835, -0.808363, 1.570796, 1.869317],accel_mss,speed_ms,0,blend_radius_m)
    |   movel([0.299698, -1.252955, -2.650962, -0.808473, 1.570796, 1.870495],accel_mss,speed_ms,0,blend_radius_m)
    |   movel([0.300787, -1.253122, -2.650872, -0.808395, 1.570796, 1.871583],accel_mss,speed_ms,0,blend_radius_m)
    |   movel([0.301875, -1.253726, -2.650547, -0.808115, 1.570796, 1.872671],accel_mss,speed_ms,0,blend_radius_m)
    |   movel([0.303062, -1.254841, -2.649947, -0.807601, 1.570796, 1.873858],accel_mss,speed_ms,0,blend_radius_m)
    |   movel([0.303576, -1.255352, -2.649672, -0.807365, 1.570796, 1.874372],accel_mss,speed_ms,0,blend_radius_m)
    |   movel([0.304570, -1.256003, -2.649320, -0.807066, 1.570796, 1.875367],accel_mss,speed_ms,0,blend_radius_m)
    |   movel([0.305115, -1.256190, -2.649219, -0.806980, 1.570796, 1.875911],accel_mss,speed_ms,0,blend_radius_m)
    |   movel([0.306798, -1.256837, -2.648869, -0.806683, 1.570796, 1.877594],accel_mss,speed_ms,0,blend_radius_m)
    |   movel([0.307267, -1.257262, -2.648639, -0.806488, 1.570796, 1.878064],accel_mss,speed_ms,0,blend_radius_m)
    |   movel([0.307601, -1.257822, -2.648335, -0.806232, 1.570796, 1.878398],accel_mss,speed_ms,0,blend_radius_m)
    |   movel([0.307826, -1.258534, -2.647948, -0.805906, 1.570796, 1.878622],accel_mss,speed_ms,0,blend_radius_m)
    |   movel([0.308075, -1.260565, -2.646843, -0.804982, 1.570796, 1.878871],accel_mss,speed_ms,0,blend_radius_m)
    |   movel([0.308074, -1.261623, -2.646264, -0.804502, 1.570796, 1.878870],accel_mss,speed_ms,0,blend_radius_m)
    |   movel([0.308211, -1.262621, -2.645718, -0.804051, 1.570796, 1.879008],accel_mss,speed_ms,0,blend_radius_m)
    |   movel([0.308440, -1.262763, -2.645639, -0.803986, 1.570796, 1.879237],accel_mss,speed_ms,0,blend_radius_m)
    |   movel([0.308766, -1.262701, -2.645673, -0.804014, 1.570796, 1.879563],accel_mss,speed_ms,0,blend_radius_m)
    |   movel([0.309063, -1.262431, -2.645821, -0.804136, 1.570796, 1.879859],accel_mss,speed_ms,0,blend_radius_m)
    |   movel([0.309238, -1.261994, -2.646061, -0.804334, 1.570796, 1.880034],accel_mss,speed_ms,0,blend_radius_m)
    |   movel([0.309308, -1.261281, -2.646451, -0.804657, 1.570796, 1.880104],accel_mss,speed_ms,0,blend_radius_m)
    |   movel([0.309051, -1.257920, -2.648282, -0.806187, 1.570796, 1.879847],accel_mss,speed_ms,0,blend_radius_m)
    |   movel([0.308534, -1.256555, -2.649022, -0.806812, 1.570796, 1.879330],accel_mss,speed_ms,0,blend_radius_m)
    |   movel([0.308137, -1.256059, -2.649290, -0.807040, 1.570796, 1.878933],accel_mss,speed_ms,0,blend_radius_m)
    |   movel([0.307627, -1.255668, -2.649501, -0.807220, 1.570796, 1.878423],accel_mss,speed_ms,0,blend_radius_m)
    |   movel([0.305525, -1.254863, -2.649935, -0.807590, 1.570796, 1.876322],accel_mss,speed_ms,0,blend_radius_m)
    |   movel([0.304976, -1.254582, -2.650087, -0.807720, 1.570796, 1.875772],accel_mss,speed_ms,0,blend_radius_m)
    |   movel([0.303851, -1.253587, -2.650622, -0.808180, 1.570796, 1.874647],accel_mss,speed_ms,0,blend_radius_m)
    |   movel([0.302807, -1.252629, -2.651136, -0.808623, 1.570796, 1.873603],accel_mss,speed_ms,0,blend_radius_m)
    |   movel([0.301797, -1.252060, -2.651441, -0.808888, 1.570796, 1.872594],accel_mss,speed_ms,0,blend_radius_m)
    |   movel([0.300725, -1.251831, -2.651564, -0.808994, 1.570796, 1.871521],accel_mss,speed_ms,0,blend_radius_m)
    |   movel([0.299508, -1.251901, -2.651527, -0.808962, 1.570796, 1.870304],accel_mss,speed_ms,0,blend_radius_m)
    |   movel([0.298229, -1.252128, -2.651405, -0.808856, 1.570796, 1.869025],accel_mss,speed_ms,0,blend_radius_m)
    |   movel([0.302359, -1.239844, -2.657895, -0.814650, 1.570796, 1.873155],accel_mss,speed_ms,0,blend_radius_m)
    |   movel([0.303065, -1.239894, -2.657869, -0.814626, 1.570796, 1.873861],accel_mss,speed_ms,0,blend_radius_m)
    |   movel([0.303826, -1.240209, -2.657705, -0.814475, 1.570796, 1.874622],accel_mss,speed_ms,0,blend_radius_m)
    |   movel([0.304470, -1.240690, -2.657454, -0.814245, 1.570796, 1.875266],accel_mss,speed_ms,0,blend_radius_m)
    |   movel([0.304977, -1.241324, -2.657123, -0.813942, 1.570796, 1.875773],accel_mss,speed_ms,0,blend_radius_m)
    |   movel([0.305731, -1.242965, -2.656263, -0.813160, 1.570796, 1.876527],accel_mss,speed_ms,0,blend_radius_m)
    |   movel([0.305931, -1.243067, -2.656210, -0.813112, 1.570796, 1.876728],accel_mss,speed_ms,0,blend_radius_m)
    |   movel([0.306599, -1.242998, -2.656246, -0.813145, 1.570796, 1.877396],accel_mss,speed_ms,0,blend_radius_m)
    |   movel([0.306868, -1.243179, -2.656151, -0.813059, 1.570796, 1.877664],accel_mss,speed_ms,0,blend_radius_m)
    |   movel([0.307015, -1.243615, -2.655922, -0.812852, 1.570796, 1.877811],accel_mss,speed_ms,0,blend_radius_m)
    |   movel([0.307047, -1.244371, -2.655524, -0.812494, 1.570796, 1.877843],accel_mss,speed_ms,0,blend_radius_m)
    |   movel([0.306779, -1.246698, -2.654296, -0.811395, 1.570796, 1.877575],accel_mss,speed_ms,0,blend_radius_m)
    |   movel([0.306008, -1.246362, -2.654474, -0.811553, 1.570796, 1.876804],accel_mss,speed_ms,0,blend_radius_m)
    |   movel([0.305318, -1.245917, -2.654709, -0.811763, 1.570796, 1.876114],accel_mss,speed_ms,0,blend_radius_m)
    |   movel([0.304476, -1.245612, -2.654870, -0.811907, 1.570796, 1.875273],accel_mss,speed_ms,0,blend_radius_m)
    |   movel([0.303527, -1.245462, -2.654949, -0.811978, 1.570796, 1.874323],accel_mss,speed_ms,0,blend_radius_m)
    |   movel([0.301828, -1.245560, -2.654897, -0.811931, 1.570796, 1.872624],accel_mss,speed_ms,0,blend_radius_m)
    |   movel([0.301456, -1.245649, -2.654851, -0.811890, 1.570796, 1.872252],accel_mss,speed_ms,0,blend_radius_m)
    |   movel([0.300973, -1.246019, -2.654655, -0.811715, 1.570796, 1.871769],accel_mss,speed_ms,0,blend_radius_m)
    |   movel([0.300752, -1.246418, -2.654444, -0.811527, 1.570796, 1.871549],accel_mss,speed_ms,0,blend_radius_m)
    |   movel([0.300798, -1.246656, -2.654318, -0.811414, 1.570796, 1.871594],accel_mss,speed_ms,0,blend_radius_m)
    |   movel([0.301157, -1.246750, -2.654269, -0.811370, 1.570796, 1.871954],accel_mss,speed_ms,0,blend_radius_m)
    |   movel([0.303060, -1.246693, -2.654298, -0.811397, 1.570796, 1.873856],accel_mss,speed_ms,0,blend_radius_m)
    |   movel([0.303582, -1.246768, -2.654259, -0.811362, 1.570796, 1.874379],accel_mss,speed_ms,0,blend_radius_m)
    |   movel([0.304671, -1.247204, -2.654028, -0.811157, 1.570796, 1.875468],accel_mss,speed_ms,0,blend_radius_m)
    |   movel([0.305226, -1.247655, -2.653789, -0.810945, 1.570796, 1.876022],accel_mss,speed_ms,0,blend_radius_m)
    |   movel([0.306298, -1.249083, -2.653031, -0.810276, 1.570796, 1.877094],accel_mss,speed_ms,0,blend_radius_m)
    |   movel([0.307038, -1.250807, -2.652112, -0.809471, 1.570796, 1.877834],accel_mss,speed_ms,0,blend_radius_m)
    |   movel([0.307251, -1.252504, -2.651203, -0.808681, 1.570796, 1.878048],accel_mss,speed_ms,0,blend_radius_m)
    |   movel([0.307296, -1.253044, -2.650914, -0.808431, 1.570796, 1.878092],accel_mss,speed_ms,0,blend_radius_m)
    |   movel([0.307475, -1.253319, -2.650766, -0.808304, 1.570796, 1.878271],accel_mss,speed_ms,0,blend_radius_m)
    |   movel([0.307768, -1.253329, -2.650761, -0.808299, 1.570796, 1.878564],accel_mss,speed_ms,0,blend_radius_m)
    |   movel([0.308145, -1.253099, -2.650884, -0.808406, 1.570796, 1.878942],accel_mss,speed_ms,0,blend_radius_m)
    |   movel([0.308338, -1.252894, -2.650994, -0.808501, 1.570796, 1.879134],accel_mss,speed_ms,0,blend_radius_m)
    |   movel([0.308506, -1.252443, -2.651236, -0.808710, 1.570796, 1.879302],accel_mss,speed_ms,0,blend_radius_m)
    |   movel([0.308518, -1.252043, -2.651450, -0.808895, 1.570796, 1.879314],accel_mss,speed_ms,0,blend_radius_m)
    |   movel([0.308278, -1.250184, -2.652444, -0.809761, 1.570796, 1.879075],accel_mss,speed_ms,0,blend_radius_m)
    |   movel([0.308018, -1.249247, -2.652943, -0.810199, 1.570796, 1.878814],accel_mss,speed_ms,0,blend_radius_m)
    |   movel([0.307457, -1.247793, -2.653716, -0.810880, 1.570796, 1.878253],accel_mss,speed_ms,0,blend_radius_m)
    |   movel([0.307484, -1.247531, -2.653855, -0.811003, 1.570796, 1.878281],accel_mss,speed_ms,0,blend_radius_m)
    |   movel([0.307860, -1.246702, -2.654294, -0.811393, 1.570796, 1.878657],accel_mss,speed_ms,0,blend_radius_m)
    |   movel([0.308096, -1.245654, -2.654848, -0.811887, 1.570796, 1.878893],accel_mss,speed_ms,0,blend_radius_m)
    |   movel([0.308312, -1.243504, -2.655980, -0.812905, 1.570796, 1.879109],accel_mss,speed_ms,0,blend_radius_m)
    |   movel([0.308227, -1.242774, -2.656363, -0.813251, 1.570796, 1.879024],accel_mss,speed_ms,0,blend_radius_m)
    |   movel([0.307995, -1.242194, -2.656667, -0.813527, 1.570796, 1.878792],accel_mss,speed_ms,0,blend_radius_m)
    |   movel([0.307659, -1.241832, -2.656857, -0.813700, 1.570796, 1.878455],accel_mss,speed_ms,0,blend_radius_m)
    |   movel([0.307258, -1.241764, -2.656892, -0.813732, 1.570796, 1.878054],accel_mss,speed_ms,0,blend_radius_m)
    |   movel([0.307070, -1.241743, -2.656903, -0.813742, 1.570796, 1.877866],accel_mss,speed_ms,0,blend_radius_m)
    |   movel([0.306530, -1.241066, -2.657258, -0.814065, 1.570796, 1.877326],accel_mss,speed_ms,0,blend_radius_m)
    |   movel([0.305977, -1.240116, -2.657754, -0.814520, 1.570796, 1.876773],accel_mss,speed_ms,0,blend_radius_m)
    |   movel([0.305186, -1.239334, -2.658161, -0.814894, 1.570796, 1.875983],accel_mss,speed_ms,0,blend_radius_m)
    |   movel([0.304251, -1.238796, -2.658441, -0.815152, 1.570796, 1.875047],accel_mss,speed_ms,0,blend_radius_m)
    |   movel([0.303267, -1.238573, -2.658557, -0.815260, 1.570796, 1.874063],accel_mss,speed_ms,0,blend_radius_m)
    |   movel([0.302793, -1.238541, -2.658573, -0.815275, 1.570796, 1.873590],accel_mss,speed_ms,0,blend_radius_m)
    |   movel([0.304551, -1.233360, -2.661249, -0.817780, 1.570796, 1.875347],accel_mss,speed_ms,0,blend_radius_m)
    |   movel([0.304863, -1.232477, -2.661702, -0.818210, 1.570796, 1.875660],accel_mss,speed_ms,0,blend_radius_m)
    |   movel([0.305199, -1.232301, -2.661792, -0.818296, 1.570796, 1.875996],accel_mss,speed_ms,0,blend_radius_m)
    |   movel([0.306515, -1.232519, -2.661680, -0.818189, 1.570796, 1.877312],accel_mss,speed_ms,0,blend_radius_m)
    |   movel([0.308530, -1.233091, -2.661387, -0.817911, 1.570796, 1.879326],accel_mss,speed_ms,0,blend_radius_m)
    |   movel([0.309553, -1.233765, -2.661041, -0.817583, 1.570796, 1.880349],accel_mss,speed_ms,0,blend_radius_m)
    |   movel([0.310420, -1.234599, -2.660612, -0.817178, 1.570796, 1.881216],accel_mss,speed_ms,0,blend_radius_m)
    |   movel([0.311088, -1.235554, -2.660120, -0.816715, 1.570796, 1.881885],accel_mss,speed_ms,0,blend_radius_m)
    |   movel([0.311565, -1.236657, -2.659550, -0.816182, 1.570796, 1.882361],accel_mss,speed_ms,0,blend_radius_m)
    |   movel([0.311829, -1.237840, -2.658937, -0.815612, 1.570796, 1.882625],accel_mss,speed_ms,0,blend_radius_m)
    |   movel([0.311898, -1.239127, -2.658269, -0.814994, 1.570796, 1.882694],accel_mss,speed_ms,0,blend_radius_m)
    |   movel([0.311758, -1.240459, -2.657574, -0.814355, 1.570796, 1.882555],accel_mss,speed_ms,0,blend_radius_m)
    |   movel([0.311409, -1.241854, -2.656845, -0.813689, 1.570796, 1.882205],accel_mss,speed_ms,0,blend_radius_m)
    |   movel([0.311125, -1.242778, -2.656361, -0.813250, 1.570796, 1.881922],accel_mss,speed_ms,0,blend_radius_m)
    |   movel([0.311020, -1.243546, -2.655958, -0.812885, 1.570796, 1.881816],accel_mss,speed_ms,0,blend_radius_m)
    |   movel([0.311138, -1.243667, -2.655894, -0.812827, 1.570796, 1.881935],accel_mss,speed_ms,0,blend_radius_m)
    |   movel([0.311454, -1.243631, -2.655913, -0.812844, 1.570796, 1.882250],accel_mss,speed_ms,0,blend_radius_m)
    |   movel([0.311640, -1.243549, -2.655956, -0.812883, 1.570796, 1.882437],accel_mss,speed_ms,0,blend_radius_m)
    |   movel([0.312027, -1.243194, -2.656143, -0.813052, 1.570796, 1.882823],accel_mss,speed_ms,0,blend_radius_m)
    |   movel([0.312216, -1.242821, -2.656339, -0.813229, 1.570796, 1.883013],accel_mss,speed_ms,0,blend_radius_m)
    |   movel([0.312711, -1.241230, -2.657172, -0.813987, 1.570796, 1.883507],accel_mss,speed_ms,0,blend_radius_m)
    |   movel([0.313116, -1.238912, -2.658381, -0.815097, 1.570796, 1.883912],accel_mss,speed_ms,0,blend_radius_m)
    |   movel([0.313017, -1.236815, -2.659468, -0.816106, 1.570796, 1.883814],accel_mss,speed_ms,0,blend_radius_m)
    |   movel([0.312398, -1.234950, -2.660431, -0.817008, 1.570796, 1.883194],accel_mss,speed_ms,0,blend_radius_m)
    |   movel([0.311260, -1.233318, -2.661271, -0.817800, 1.570796, 1.882057],accel_mss,speed_ms,0,blend_radius_m)
    |   movel([0.310181, -1.232378, -2.661753, -0.818258, 1.570796, 1.880977],accel_mss,speed_ms,0,blend_radius_m)
    |   movel([0.308952, -1.231727, -2.662086, -0.818576, 1.570796, 1.879749],accel_mss,speed_ms,0,blend_radius_m)
    |   movel([0.307490, -1.231331, -2.662289, -0.818769, 1.570796, 1.878287],accel_mss,speed_ms,0,blend_radius_m)
    |   movel([0.305711, -1.231164, -2.662374, -0.818851, 1.570796, 1.876507],accel_mss,speed_ms,0,blend_radius_m)
    |   movel([0.305154, -1.231147, -2.662383, -0.818859, 1.570796, 1.875950],accel_mss,speed_ms,0,blend_radius_m)
    |   movel([0.307724, -1.223792, -2.666109, -0.822488, 1.570796, 1.878520],accel_mss,speed_ms,0,blend_radius_m)
    |   movel([0.308064, -1.222715, -2.666649, -0.823024, 1.570796, 1.878860],accel_mss,speed_ms,0,blend_radius_m)
    |   movel([0.310823, -1.222741, -2.666636, -0.823011, 1.570796, 1.881619],accel_mss,speed_ms,0,blend_radius_m)
    |   movel([0.312235, -1.223117, -2.666448, -0.822824, 1.570796, 1.883032],accel_mss,speed_ms,0,blend_radius_m)
    |   movel([0.313426, -1.223781, -2.666115, -0.822493, 1.570796, 1.884222],accel_mss,speed_ms,0,blend_radius_m)
    |   movel([0.314360, -1.224713, -2.665646, -0.822030, 1.570796, 1.885157],accel_mss,speed_ms,0,blend_radius_m)
    |   movel([0.315060, -1.225944, -2.665025, -0.821420, 1.570796, 1.885856],accel_mss,speed_ms,0,blend_radius_m)
    |   movel([0.315470, -1.227376, -2.664301, -0.820712, 1.570796, 1.886267],accel_mss,speed_ms,0,blend_radius_m)
    |   movel([0.315622, -1.229098, -2.663427, -0.819864, 1.570796, 1.886419],accel_mss,speed_ms,0,blend_radius_m)
    |   movel([0.315517, -1.230933, -2.662492, -0.818964, 1.570796, 1.886314],accel_mss,speed_ms,0,blend_radius_m)
    |   movel([0.315016, -1.233646, -2.661102, -0.817640, 1.570796, 1.885813],accel_mss,speed_ms,0,blend_radius_m)
    |   movel([0.314883, -1.234232, -2.660801, -0.817356, 1.570796, 1.885680],accel_mss,speed_ms,0,blend_radius_m)
    |   movel([0.314937, -1.234616, -2.660604, -0.817170, 1.570796, 1.885733],accel_mss,speed_ms,0,blend_radius_m)
    |   movel([0.315162, -1.234759, -2.660530, -0.817100, 1.570796, 1.885958],accel_mss,speed_ms,0,blend_radius_m)
    |   movel([0.315524, -1.234680, -2.660571, -0.817139, 1.570796, 1.886320],accel_mss,speed_ms,0,blend_radius_m)
    |   movel([0.315834, -1.234395, -2.660717, -0.817277, 1.570796, 1.886630],accel_mss,speed_ms,0,blend_radius_m)
    |   movel([0.316098, -1.233847, -2.660999, -0.817543, 1.570796, 1.886894],accel_mss,speed_ms,0,blend_radius_m)
    |   movel([0.316346, -1.232992, -2.661438, -0.817959, 1.570796, 1.887142],accel_mss,speed_ms,0,blend_radius_m)
    |   movel([0.316853, -1.229869, -2.663035, -0.819485, 1.570796, 1.887650],accel_mss,speed_ms,0,blend_radius_m)
    |   movel([0.316917, -1.228157, -2.663905, -0.820327, 1.570796, 1.887713],accel_mss,speed_ms,0,blend_radius_m)
    |   movel([0.316790, -1.226696, -2.664645, -0.821048, 1.570796, 1.887587],accel_mss,speed_ms,0,blend_radius_m)
    |   movel([0.316447, -1.225354, -2.665323, -0.821712, 1.570796, 1.887243],accel_mss,speed_ms,0,blend_radius_m)
    |   movel([0.315923, -1.224231, -2.665889, -0.822270, 1.570796, 1.886719],accel_mss,speed_ms,0,blend_radius_m)
    |   movel([0.315190, -1.223275, -2.666369, -0.822745, 1.570796, 1.885987],accel_mss,speed_ms,0,blend_radius_m)
    |   movel([0.314272, -1.222502, -2.666756, -0.823131, 1.570796, 1.885068],accel_mss,speed_ms,0,blend_radius_m)
    |   movel([0.313173, -1.221930, -2.667043, -0.823416, 1.570796, 1.883969],accel_mss,speed_ms,0,blend_radius_m)
    |   movel([0.311152, -1.221458, -2.667279, -0.823652, 1.570796, 1.881948],accel_mss,speed_ms,0,blend_radius_m)
    |   movel([0.310058, -1.221390, -2.667313, -0.823686, 1.570796, 1.880855],accel_mss,speed_ms,0,blend_radius_m)
    |   movel([0.308780, -1.221519, -2.667248, -0.823622, 1.570796, 1.879576],accel_mss,speed_ms,0,blend_radius_m)
    |   movel([0.308576, -1.221490, -2.667263, -0.823636, 1.570796, 1.879372],accel_mss,speed_ms,0,blend_radius_m)
    |   movel([0.308476, -1.221150, -2.667433, -0.823806, 1.570796, 1.879272],accel_mss,speed_ms,0,blend_radius_m)
    |   movel([0.308540, -1.220819, -2.667598, -0.823972, 1.570796, 1.879336],accel_mss,speed_ms,0,blend_radius_m)
    |   movel([0.311033, -1.212080, -2.671916, -0.828394, 1.570796, 1.881829],accel_mss,speed_ms,0,blend_radius_m)
    |   movel([0.311437, -1.210596, -2.672640, -0.829153, 1.570796, 1.882233],accel_mss,speed_ms,0,blend_radius_m)
    |   movel([0.311738, -1.209404, -2.673221, -0.829765, 1.570796, 1.882534],accel_mss,speed_ms,0,blend_radius_m)
    |   movel([0.311912, -1.209245, -2.673298, -0.829846, 1.570796, 1.882708],accel_mss,speed_ms,0,blend_radius_m)
    |   movel([0.312802, -1.208918, -2.673457, -0.830015, 1.570796, 1.883599],accel_mss,speed_ms,0,blend_radius_m)
    |   movel([0.313320, -1.208887, -2.673472, -0.830030, 1.570796, 1.884116],accel_mss,speed_ms,0,blend_radius_m)
    |   movel([0.315123, -1.209132, -2.673353, -0.829904, 1.570796, 1.885919],accel_mss,speed_ms,0,blend_radius_m)
    |   movel([0.316823, -1.209570, -2.673140, -0.829679, 1.570796, 1.887620],accel_mss,speed_ms,0,blend_radius_m)
    |   movel([0.317646, -1.210121, -2.672872, -0.829397, 1.570796, 1.888442],accel_mss,speed_ms,0,blend_radius_m)
    |   movel([0.317833, -1.210446, -2.672713, -0.829230, 1.570796, 1.888629],accel_mss,speed_ms,0,blend_radius_m)
    |   movel([0.318583, -1.213403, -2.671267, -0.827719, 1.570796, 1.889379],accel_mss,speed_ms,0,blend_radius_m)
    |   movel([0.318824, -1.214201, -2.670876, -0.827313, 1.570796, 1.889620],accel_mss,speed_ms,0,blend_radius_m)
    |   movel([0.319444, -1.215472, -2.670250, -0.826667, 1.570796, 1.890240],accel_mss,speed_ms,0,blend_radius_m)
    |   movel([0.320317, -1.217024, -2.669484, -0.825882, 1.570796, 1.891114],accel_mss,speed_ms,0,blend_radius_m)
    |   movel([0.320605, -1.218352, -2.668826, -0.825212, 1.570796, 1.891401],accel_mss,speed_ms,0,blend_radius_m)
    |   movel([0.320411, -1.220048, -2.667982, -0.824359, 1.570796, 1.891207],accel_mss,speed_ms,0,blend_radius_m)
    |   movel([0.319634, -1.222979, -2.666517, -0.822893, 1.570796, 1.890430],accel_mss,speed_ms,0,blend_radius_m)
    |   movel([0.318629, -1.226389, -2.664800, -0.821199, 1.570796, 1.889426],accel_mss,speed_ms,0,blend_radius_m)
    |   movel([0.319172, -1.226361, -2.664815, -0.821213, 1.570796, 1.889969],accel_mss,speed_ms,0,blend_radius_m)
    |   movel([0.319713, -1.226330, -2.664830, -0.821229, 1.570796, 1.890510],accel_mss,speed_ms,0,blend_radius_m)
    |   movel([0.321495, -1.220530, -2.667742, -0.824117, 1.570796, 1.892292],accel_mss,speed_ms,0,blend_radius_m)
    |   movel([0.321734, -1.219379, -2.668315, -0.824695, 1.570796, 1.892530],accel_mss,speed_ms,0,blend_radius_m)
    |   movel([0.321811, -1.217362, -2.669316, -0.825711, 1.570796, 1.892607],accel_mss,speed_ms,0,blend_radius_m)
    |   movel([0.321631, -1.216533, -2.669726, -0.826130, 1.570796, 1.892428],accel_mss,speed_ms,0,blend_radius_m)
    |   movel([0.320456, -1.214180, -2.670886, -0.827323, 1.570796, 1.891252],accel_mss,speed_ms,0,blend_radius_m)
    |   movel([0.320144, -1.213447, -2.671246, -0.827696, 1.570796, 1.890940],accel_mss,speed_ms,0,blend_radius_m)
    |   movel([0.319421, -1.210368, -2.672751, -0.829270, 1.570796, 1.890218],accel_mss,speed_ms,0,blend_radius_m)
    |   movel([0.319032, -1.209396, -2.673224, -0.829769, 1.570796, 1.889828],accel_mss,speed_ms,0,blend_radius_m)
    |   movel([0.318498, -1.208738, -2.673544, -0.830107, 1.570796, 1.889294],accel_mss,speed_ms,0,blend_radius_m)
    |   movel([0.317774, -1.208297, -2.673758, -0.830334, 1.570796, 1.888570],accel_mss,speed_ms,0,blend_radius_m)
    |   movel([0.316818, -1.208009, -2.673898, -0.830483, 1.570796, 1.887615],accel_mss,speed_ms,0,blend_radius_m)
    |   movel([0.315527, -1.207777, -2.674010, -0.830602, 1.570796, 1.886323],accel_mss,speed_ms,0,blend_radius_m)
    |   movel([0.313141, -1.207636, -2.674078, -0.830675, 1.570796, 1.883937],accel_mss,speed_ms,0,blend_radius_m)
    |   movel([0.312138, -1.207707, -2.674044, -0.830638, 1.570796, 1.882934],accel_mss,speed_ms,0,blend_radius_m)
    |   movel([0.313556, -1.200426, -2.677540, -0.834423, 1.570796, 1.884353],accel_mss,speed_ms,0,blend_radius_m)
    |   movel([0.313840, -1.198856, -2.678286, -0.835246, 1.570796, 1.884637],accel_mss,speed_ms,0,blend_radius_m)
    |   movel([0.314179, -1.197738, -2.678816, -0.835835, 1.570796, 1.884975],accel_mss,speed_ms,0,blend_radius_m)
    |   movel([0.314601, -1.196918, -2.679204, -0.836267, 1.570796, 1.885398],accel_mss,speed_ms,0,blend_radius_m)
    |   movel([0.315151, -1.196305, -2.679493, -0.836591, 1.570796, 1.885947],accel_mss,speed_ms,0,blend_radius_m)
    |   movel([0.315908, -1.195813, -2.679725, -0.836851, 1.570796, 1.886705],accel_mss,speed_ms,0,blend_radius_m)
    |   movel([0.316676, -1.195544, -2.679852, -0.836993, 1.570796, 1.887472],accel_mss,speed_ms,0,blend_radius_m)
    |   movel([0.317657, -1.195428, -2.679906, -0.837055, 1.570796, 1.888453],accel_mss,speed_ms,0,blend_radius_m)
    |   movel([0.319555, -1.195658, -2.679798, -0.836933, 1.570796, 1.890351],accel_mss,speed_ms,0,blend_radius_m)
    |   movel([0.320437, -1.196004, -2.679635, -0.836750, 1.570796, 1.891233],accel_mss,speed_ms,0,blend_radius_m)
    |   movel([0.321877, -1.197120, -2.679109, -0.836161, 1.570796, 1.892673],accel_mss,speed_ms,0,blend_radius_m)
    |   movel([0.322422, -1.197652, -2.678857, -0.835880, 1.570796, 1.893219],accel_mss,speed_ms,0,blend_radius_m)
    |   movel([0.322861, -1.197801, -2.678786, -0.835802, 1.570796, 1.893657],accel_mss,speed_ms,0,blend_radius_m)
    |   movel([0.323260, -1.197629, -2.678868, -0.835892, 1.570796, 1.894056],accel_mss,speed_ms,0,blend_radius_m)
    |   movel([0.323887, -1.196842, -2.679239, -0.836307, 1.570796, 1.894683],accel_mss,speed_ms,0,blend_radius_m)
    |   movel([0.324347, -1.196713, -2.679300, -0.836375, 1.570796, 1.895143],accel_mss,speed_ms,0,blend_radius_m)
    |   movel([0.324516, -1.196869, -2.679227, -0.836293, 1.570796, 1.895313],accel_mss,speed_ms,0,blend_radius_m)
    |   movel([0.325594, -1.199811, -2.677833, -0.834745, 1.570796, 1.896390],accel_mss,speed_ms,0,blend_radius_m)
    |   movel([0.325735, -1.201060, -2.677238, -0.834091, 1.570796, 1.896532],accel_mss,speed_ms,0,blend_radius_m)
    |   movel([0.325637, -1.202734, -2.676438, -0.833217, 1.570796, 1.896433],accel_mss,speed_ms,0,blend_radius_m)
    |   movel([0.325356, -1.204495, -2.675593, -0.832300, 1.570796, 1.896153],accel_mss,speed_ms,0,blend_radius_m)
    |   movel([0.324074, -1.209177, -2.673330, -0.829881, 1.570796, 1.894870],accel_mss,speed_ms,0,blend_radius_m)
    |   movel([0.322863, -1.213000, -2.671465, -0.827924, 1.570796, 1.893659],accel_mss,speed_ms,0,blend_radius_m)
    |   movel([0.323625, -1.212826, -2.671550, -0.828013, 1.570796, 1.894421],accel_mss,speed_ms,0,blend_radius_m)
    |   movel([0.323837, -1.212667, -2.671628, -0.828094, 1.570796, 1.894633],accel_mss,speed_ms,0,blend_radius_m)
    |   movel([0.324326, -1.211845, -2.672030, -0.828513, 1.570796, 1.895123],accel_mss,speed_ms,0,blend_radius_m)
    |   movel([0.324942, -1.210344, -2.672763, -0.829282, 1.570796, 1.895738],accel_mss,speed_ms,0,blend_radius_m)
    |   movel([0.325733, -1.207692, -2.674051, -0.830646, 1.570796, 1.896530],accel_mss,speed_ms,0,blend_radius_m)
    |   movel([0.326441, -1.204978, -2.675361, -0.832050, 1.570796, 1.897237],accel_mss,speed_ms,0,blend_radius_m)
    |   movel([0.326801, -1.203042, -2.676291, -0.833056, 1.570796, 1.897597],accel_mss,speed_ms,0,blend_radius_m)
    |   movel([0.326967, -1.201288, -2.677129, -0.833972, 1.570796, 1.897763],accel_mss,speed_ms,0,blend_radius_m)
    |   movel([0.326964, -1.199908, -2.677787, -0.834695, 1.570796, 1.897761],accel_mss,speed_ms,0,blend_radius_m)
    |   movel([0.326783, -1.198679, -2.678370, -0.835339, 1.570796, 1.897579],accel_mss,speed_ms,0,blend_radius_m)
    |   movel([0.326400, -1.197399, -2.678976, -0.836013, 1.570796, 1.897197],accel_mss,speed_ms,0,blend_radius_m)
    |   movel([0.325886, -1.196287, -2.679502, -0.836600, 1.570796, 1.896682],accel_mss,speed_ms,0,blend_radius_m)
    |   movel([0.325314, -1.195649, -2.679802, -0.836938, 1.570796, 1.896110],accel_mss,speed_ms,0,blend_radius_m)
    |   movel([0.324665, -1.195434, -2.679904, -0.837052, 1.570796, 1.895461],accel_mss,speed_ms,0,blend_radius_m)
    |   movel([0.323510, -1.195767, -2.679747, -0.836875, 1.570796, 1.894306],accel_mss,speed_ms,0,blend_radius_m)
    |   movel([0.323189, -1.195777, -2.679742, -0.836870, 1.570796, 1.893985],accel_mss,speed_ms,0,blend_radius_m)
    |   movel([0.322217, -1.195220, -2.680004, -0.837165, 1.570796, 1.893014],accel_mss,speed_ms,0,blend_radius_m)
    |   movel([0.320536, -1.194391, -2.680394, -0.837604, 1.570796, 1.891333],accel_mss,speed_ms,0,blend_radius_m)
    |   movel([0.319626, -1.194178, -2.680494, -0.837717, 1.570796, 1.890423],accel_mss,speed_ms,0,blend_radius_m)
    |   movel([0.318635, -1.194106, -2.680528, -0.837755, 1.570796, 1.889431],accel_mss,speed_ms,0,blend_radius_m)
    |   movel([0.316748, -1.194381, -2.680398, -0.837609, 1.570796, 1.887545],accel_mss,speed_ms,0,blend_radius_m)
    |   movel([0.315928, -1.194701, -2.680248, -0.837440, 1.570796, 1.886724],accel_mss,speed_ms,0,blend_radius_m)
    |   movel([0.314150, -1.195850, -2.679708, -0.836832, 1.570796, 1.884947],accel_mss,speed_ms,0,blend_radius_m)
    |   movel([0.314093, -1.194358, -2.680410, -0.837622, 1.570796, 1.884889],accel_mss,speed_ms,0,blend_radius_m)
    |   movel([0.313895, -1.191852, -2.681583, -0.838954, 1.570796, 1.884691],accel_mss,speed_ms,0,blend_radius_m)
    |   movel([0.313298, -1.189575, -2.682643, -0.840171, 1.570796, 1.884094],accel_mss,speed_ms,0,blend_radius_m)
    |   movel([0.312303, -1.187561, -2.683576, -0.841252, 1.570796, 1.883099],accel_mss,speed_ms,0,blend_radius_m)
    |   movel([0.310930, -1.185860, -2.684360, -0.842169, 1.570796, 1.881726],accel_mss,speed_ms,0,blend_radius_m)
    |   movel([0.309157, -1.184460, -2.685004, -0.842925, 1.570796, 1.879954],accel_mss,speed_ms,0,blend_radius_m)
    |   movel([0.307063, -1.183430, -2.685476, -0.843483, 1.570796, 1.877859],accel_mss,speed_ms,0,blend_radius_m)
    |   movel([0.304582, -1.182735, -2.685794, -0.843860, 1.570796, 1.875378],accel_mss,speed_ms,0,blend_radius_m)
    |   movel([0.301870, -1.182412, -2.685941, -0.844036, 1.570796, 1.872666],accel_mss,speed_ms,0,blend_radius_m)
    |   movel([0.299054, -1.182450, -2.685924, -0.844015, 1.570796, 1.869850],accel_mss,speed_ms,0,blend_radius_m)
    |   movel([0.296092, -1.182837, -2.685747, -0.843805, 1.570796, 1.866888],accel_mss,speed_ms,0,blend_radius_m)
    |   movel([0.293103, -1.183557, -2.685418, -0.843414, 1.570796, 1.863899],accel_mss,speed_ms,0,blend_radius_m)
    |   movel([0.290039, -1.184626, -2.684928, -0.842835, 1.570796, 1.860835],accel_mss,speed_ms,0,blend_radius_m)
    |   movel([0.287095, -1.185967, -2.684311, -0.842111, 1.570796, 1.857892],accel_mss,speed_ms,0,blend_radius_m)
    |   movel([0.284170, -1.187615, -2.683551, -0.841223, 1.570796, 1.854967],accel_mss,speed_ms,0,blend_radius_m)
    |   movel([0.281478, -1.189461, -2.682695, -0.840232, 1.570796, 1.852275],accel_mss,speed_ms,0,blend_radius_m)
    |   movel([0.278920, -1.191575, -2.681712, -0.839102, 1.570796, 1.849717],accel_mss,speed_ms,0,blend_radius_m)
    |   movel([0.278147, -1.192201, -2.681420, -0.838768, 1.570796, 1.848943],accel_mss,speed_ms,0,blend_radius_m)
    |   movel([0.277595, -1.192452, -2.681303, -0.838635, 1.570796, 1.848392],accel_mss,speed_ms,0,blend_radius_m)
    |   movel([0.277088, -1.192417, -2.681319, -0.838653, 1.570796, 1.847885],accel_mss,speed_ms,0,blend_radius_m)
    |   movel([0.276430, -1.192064, -2.681484, -0.838841, 1.570796, 1.847227],accel_mss,speed_ms,0,blend_radius_m)
    |   movel([0.275920, -1.191539, -2.681729, -0.839121, 1.570796, 1.846716],accel_mss,speed_ms,0,blend_radius_m)
    |   movel([0.275657, -1.190814, -2.682067, -0.839508, 1.570796, 1.846453],accel_mss,speed_ms,0,blend_radius_m)
    |   movel([0.275650, -1.189893, -2.682495, -0.840001, 1.570796, 1.846446],accel_mss,speed_ms,0,blend_radius_m)
    |   movel([0.276346, -1.187175, -2.683754, -0.841460, 1.570796, 1.847142],accel_mss,speed_ms,0,blend_radius_m)
    |   movel([0.276292, -1.187004, -2.683833, -0.841552, 1.570796, 1.847088],accel_mss,speed_ms,0,blend_radius_m)
    |   movel([0.275981, -1.186928, -2.683868, -0.841593, 1.570796, 1.846777],accel_mss,speed_ms,0,blend_radius_m)
    |   movel([0.275931, -1.186702, -2.683973, -0.841715, 1.570796, 1.846727],accel_mss,speed_ms,0,blend_radius_m)
    |   movel([0.276054, -1.185635, -2.684464, -0.842290, 1.570796, 1.846850],accel_mss,speed_ms,0,blend_radius_m)
    |   movel([0.276410, -1.184076, -2.685180, -0.843133, 1.570796, 1.847206],accel_mss,speed_ms,0,blend_radius_m)
    |   movel([0.276896, -1.182702, -2.685809, -0.843878, 1.570796, 1.847692],accel_mss,speed_ms,0,blend_radius_m)
    |   movel([0.277562, -1.181372, -2.686416, -0.844601, 1.570796, 1.848358],accel_mss,speed_ms,0,blend_radius_m)
    |   movel([0.279147, -1.178978, -2.687503, -0.845908, 1.570796, 1.849943],accel_mss,speed_ms,0,blend_radius_m)
    |   movel([0.279438, -1.178486, -2.687726, -0.846177, 1.570796, 1.850234],accel_mss,speed_ms,0,blend_radius_m)
    |   movel([0.279463, -1.177984, -2.687953, -0.846452, 1.570796, 1.850259],accel_mss,speed_ms,0,blend_radius_m)
    |   movel([0.279118, -1.177897, -2.687992, -0.846500, 1.570796, 1.849914],accel_mss,speed_ms,0,blend_radius_m)
    |   movel([0.278679, -1.178131, -2.687887, -0.846371, 1.570796, 1.849476],accel_mss,speed_ms,0,blend_radius_m)
    |   movel([0.278077, -1.178795, -2.687586, -0.846008, 1.570796, 1.848873],accel_mss,speed_ms,0,blend_radius_m)
    |   movel([0.276506, -1.181103, -2.686538, -0.844748, 1.570796, 1.847302],accel_mss,speed_ms,0,blend_radius_m)
    |   movel([0.276053, -1.181914, -2.686168, -0.844306, 1.570796, 1.846849],accel_mss,speed_ms,0,blend_radius_m)
    |   movel([0.275296, -1.183840, -2.685288, -0.843261, 1.570796, 1.846092],accel_mss,speed_ms,0,blend_radius_m)
    |   movel([0.274880, -1.185276, -2.684629, -0.842484, 1.570796, 1.845676],accel_mss,speed_ms,0,blend_radius_m)
    |   movel([0.274671, -1.186469, -2.684080, -0.841840, 1.570796, 1.845468],accel_mss,speed_ms,0,blend_radius_m)
    |   movel([0.274657, -1.187302, -2.683695, -0.841391, 1.570796, 1.845453],accel_mss,speed_ms,0,blend_radius_m)
    |   movel([0.275027, -1.187513, -2.683598, -0.841278, 1.570796, 1.845823],accel_mss,speed_ms,0,blend_radius_m)
    |   movel([0.275025, -1.187754, -2.683487, -0.841148, 1.570796, 1.845821],accel_mss,speed_ms,0,blend_radius_m)
    |   movel([0.274646, -1.189036, -2.682893, -0.840460, 1.570796, 1.845442],accel_mss,speed_ms,0,blend_radius_m)
    |   movel([0.274361, -1.189941, -2.682473, -0.839975, 1.570796, 1.845157],accel_mss,speed_ms,0,blend_radius_m)
    |   movel([0.274212, -1.191020, -2.681970, -0.839398, 1.570796, 1.845008],accel_mss,speed_ms,0,blend_radius_m)
    |   movel([0.274288, -1.191546, -2.681726, -0.839118, 1.570796, 1.845085],accel_mss,speed_ms,0,blend_radius_m)
    |   movel([0.275011, -1.192839, -2.681121, -0.838429, 1.570796, 1.845808],accel_mss,speed_ms,0,blend_radius_m)
    |   movel([0.275594, -1.193429, -2.680845, -0.838115, 1.570796, 1.846390],accel_mss,speed_ms,0,blend_radius_m)
    |   movel([0.276283, -1.193909, -2.680620, -0.837860, 1.570796, 1.847079],accel_mss,speed_ms,0,blend_radius_m)
    |   movel([0.276249, -1.194098, -2.680531, -0.837760, 1.570796, 1.847045],accel_mss,speed_ms,0,blend_radius_m)
    |   movel([0.273944, -1.196974, -2.679177, -0.836238, 1.570796, 1.844740],accel_mss,speed_ms,0,blend_radius_m)
    |   movel([0.272645, -1.198832, -2.678298, -0.835260, 1.570796, 1.843441],accel_mss,speed_ms,0,blend_radius_m)
    |   movel([0.271439, -1.200820, -2.677352, -0.834217, 1.570796, 1.842235],accel_mss,speed_ms,0,blend_radius_m)
    |   movel([0.270389, -1.202820, -2.676397, -0.833172, 1.570796, 1.841186],accel_mss,speed_ms,0,blend_radius_m)
    |   movel([0.269450, -1.204938, -2.675380, -0.832071, 1.570796, 1.840246],accel_mss,speed_ms,0,blend_radius_m)
    |   movel([0.268680, -1.207032, -2.674370, -0.830987, 1.570796, 1.839476],accel_mss,speed_ms,0,blend_radius_m)
    |   movel([0.268040, -1.209214, -2.673313, -0.829862, 1.570796, 1.838837],accel_mss,speed_ms,0,blend_radius_m)
    |   movel([0.267559, -1.211351, -2.672272, -0.828766, 1.570796, 1.838355],accel_mss,speed_ms,0,blend_radius_m)
    |   movel([0.266982, -1.215137, -2.670415, -0.826837, 1.570796, 1.837779],accel_mss,speed_ms,0,blend_radius_m)
    |   movel([0.266864, -1.216758, -2.669615, -0.826016, 1.570796, 1.837660],accel_mss,speed_ms,0,blend_radius_m)
    |   movel([0.266768, -1.219873, -2.668069, -0.824447, 1.570796, 1.837564],accel_mss,speed_ms,0,blend_radius_m)
    |   movel([0.266631, -1.220170, -2.667921, -0.824297, 1.570796, 1.837427],accel_mss,speed_ms,0,blend_radius_m)
    |   movel([0.266015, -1.220944, -2.667536, -0.823910, 1.570796, 1.836812],accel_mss,speed_ms,0,blend_radius_m)
    |   movel([0.265842, -1.221404, -2.667306, -0.823680, 1.570796, 1.836638],accel_mss,speed_ms,0,blend_radius_m)
    |   movel([0.265786, -1.222654, -2.666680, -0.823055, 1.570796, 1.836582],accel_mss,speed_ms,0,blend_radius_m)
    |   movel([0.266140, -1.224026, -2.665992, -0.822371, 1.570796, 1.836936],accel_mss,speed_ms,0,blend_radius_m)
    |   movel([0.267363, -1.226122, -2.664935, -0.821332, 1.570796, 1.838159],accel_mss,speed_ms,0,blend_radius_m)
    |   movel([0.267481, -1.226485, -2.664752, -0.821152, 1.570796, 1.838277],accel_mss,speed_ms,0,blend_radius_m)
    |   movel([0.267375, -1.227447, -2.664265, -0.820677, 1.570796, 1.838171],accel_mss,speed_ms,0,blend_radius_m)
    |   movel([0.267453, -1.228475, -2.663744, -0.820170, 1.570796, 1.838249],accel_mss,speed_ms,0,blend_radius_m)
    |   movel([0.267931, -1.230345, -2.662792, -0.819252, 1.570796, 1.838727],accel_mss,speed_ms,0,blend_radius_m)
    |   movel([0.268140, -1.230904, -2.662507, -0.818978, 1.570796, 1.838936],accel_mss,speed_ms,0,blend_radius_m)
    |   movel([0.268194, -1.232056, -2.661918, -0.818415, 1.570796, 1.838990],accel_mss,speed_ms,0,blend_radius_m)
    |   movel([0.268045, -1.233067, -2.661400, -0.817922, 1.570796, 1.838841],accel_mss,speed_ms,0,blend_radius_m)
    |   movel([0.267477, -1.235473, -2.660162, -0.816755, 1.570796, 1.838273],accel_mss,speed_ms,0,blend_radius_m)
    |   movel([0.267043, -1.236661, -2.659548, -0.816180, 1.570796, 1.837839],accel_mss,speed_ms,0,blend_radius_m)
    |   movel([0.266098, -1.238791, -2.658443, -0.815155, 1.570796, 1.836895],accel_mss,speed_ms,0,blend_radius_m)
    |   movel([0.265917, -1.239065, -2.658301, -0.815023, 1.570796, 1.836713],accel_mss,speed_ms,0,blend_radius_m)
    |   movel([0.265496, -1.239210, -2.658225, -0.814954, 1.570796, 1.836292],accel_mss,speed_ms,0,blend_radius_m)
    |   movel([0.264587, -1.239222, -2.658219, -0.814948, 1.570796, 1.835383],accel_mss,speed_ms,0,blend_radius_m)
    |   movel([0.263337, -1.239425, -2.658113, -0.814850, 1.570796, 1.834133],accel_mss,speed_ms,0,blend_radius_m)
    |   movel([0.262051, -1.239745, -2.657947, -0.814697, 1.570796, 1.832848],accel_mss,speed_ms,0,blend_radius_m)
    |   movel([0.261042, -1.240125, -2.657749, -0.814515, 1.570796, 1.831838],accel_mss,speed_ms,0,blend_radius_m)
    |   movel([0.260123, -1.240632, -2.657484, -0.814273, 1.570796, 1.830919],accel_mss,speed_ms,0,blend_radius_m)
    |   movel([0.259205, -1.241297, -2.657137, -0.813955, 1.570796, 1.830001],accel_mss,speed_ms,0,blend_radius_m)
    |   movel([0.258433, -1.242002, -2.656768, -0.813619, 1.570796, 1.829230],accel_mss,speed_ms,0,blend_radius_m)
    |   movel([0.257749, -1.242926, -2.656284, -0.813179, 1.570796, 1.828545],accel_mss,speed_ms,0,blend_radius_m)
    |   movel([0.257345, -1.242984, -2.656253, -0.813152, 1.570796, 1.828141],accel_mss,speed_ms,0,blend_radius_m)
    |   movel([0.256669, -1.240594, -2.657504, -0.814291, 1.570796, 1.827465],accel_mss,speed_ms,0,blend_radius_m)
    |   movel([0.255567, -1.235985, -2.659897, -0.816507, 1.570796, 1.826363],accel_mss,speed_ms,0,blend_radius_m)
    |   movel([0.255335, -1.234706, -2.660557, -0.817126, 1.570796, 1.826131],accel_mss,speed_ms,0,blend_radius_m)
    |   movel([0.255383, -1.233841, -2.661002, -0.817546, 1.570796, 1.826180],accel_mss,speed_ms,0,blend_radius_m)
    |   movel([0.255609, -1.233567, -2.661143, -0.817679, 1.570796, 1.826405],accel_mss,speed_ms,0,blend_radius_m)
    |   movel([0.256221, -1.233142, -2.661361, -0.817886, 1.570796, 1.827018],accel_mss,speed_ms,0,blend_radius_m)
    |   movel([0.256861, -1.232818, -2.661528, -0.818044, 1.570796, 1.827658],accel_mss,speed_ms,0,blend_radius_m)
    |   movel([0.258432, -1.232316, -2.661785, -0.818288, 1.570796, 1.829229],accel_mss,speed_ms,0,blend_radius_m)
    |   movel([0.260030, -1.232123, -2.661884, -0.818383, 1.570796, 1.830826],accel_mss,speed_ms,0,blend_radius_m)
    |   movel([0.261369, -1.232298, -2.661794, -0.818297, 1.570796, 1.832165],accel_mss,speed_ms,0,blend_radius_m)
    |   movel([0.262599, -1.232916, -2.661477, -0.817996, 1.570796, 1.833395],accel_mss,speed_ms,0,blend_radius_m)
    |   movel([0.263593, -1.233953, -2.660945, -0.817492, 1.570796, 1.834389],accel_mss,speed_ms,0,blend_radius_m)
    |   movel([0.264241, -1.235257, -2.660273, -0.816859, 1.570796, 1.835037],accel_mss,speed_ms,0,blend_radius_m)
    |   movel([0.264438, -1.236668, -2.659544, -0.816177, 1.570796, 1.835234],accel_mss,speed_ms,0,blend_radius_m)
    |   movel([0.264450, -1.237143, -2.659298, -0.815947, 1.570796, 1.835246],accel_mss,speed_ms,0,blend_radius_m)
    |   movel([0.264683, -1.237476, -2.659126, -0.815787, 1.570796, 1.835479],accel_mss,speed_ms,0,blend_radius_m)
    |   movel([0.264976, -1.237485, -2.659121, -0.815783, 1.570796, 1.835772],accel_mss,speed_ms,0,blend_radius_m)
    |   movel([0.265472, -1.237327, -2.659203, -0.815859, 1.570796, 1.836268],accel_mss,speed_ms,0,blend_radius_m)
    |   movel([0.265556, -1.237139, -2.659301, -0.815950, 1.570796, 1.836352],accel_mss,speed_ms,0,blend_radius_m)
    |   movel([0.265671, -1.235678, -2.660056, -0.816655, 1.570796, 1.836467],accel_mss,speed_ms,0,blend_radius_m)
    |   movel([0.265548, -1.234849, -2.660483, -0.817056, 1.570796, 1.836344],accel_mss,speed_ms,0,blend_radius_m)
    |   movel([0.264840, -1.233206, -2.661329, -0.817855, 1.570796, 1.835636],accel_mss,speed_ms,0,blend_radius_m)
    |   movel([0.263647, -1.231876, -2.662010, -0.818503, 1.570796, 1.834443],accel_mss,speed_ms,0,blend_radius_m)
    |   movel([0.262931, -1.231416, -2.662245, -0.818728, 1.570796, 1.833727],accel_mss,speed_ms,0,blend_radius_m)
    |   movel([0.262111, -1.231087, -2.662413, -0.818889, 1.570796, 1.832907],accel_mss,speed_ms,0,blend_radius_m)
    |   movel([0.260872, -1.230878, -2.662520, -0.818991, 1.570796, 1.831669],accel_mss,speed_ms,0,blend_radius_m)
    |   movel([0.259459, -1.230939, -2.662489, -0.818961, 1.570796, 1.830255],accel_mss,speed_ms,0,blend_radius_m)
    |   movel([0.258021, -1.231253, -2.662328, -0.818807, 1.570796, 1.828817],accel_mss,speed_ms,0,blend_radius_m)
    |   movel([0.256718, -1.231798, -2.662050, -0.818541, 1.570796, 1.827514],accel_mss,speed_ms,0,blend_radius_m)
    |   movel([0.255171, -1.232564, -2.661657, -0.818167, 1.570796, 1.825967],accel_mss,speed_ms,0,blend_radius_m)
    |   movel([0.255001, -1.232517, -2.661682, -0.818190, 1.570796, 1.825797],accel_mss,speed_ms,0,blend_radius_m)
    |   movel([0.254625, -1.229815, -2.663062, -0.819512, 1.570796, 1.825421],accel_mss,speed_ms,0,blend_radius_m)
    |   movel([0.254447, -1.228508, -2.663727, -0.820154, 1.570796, 1.825243],accel_mss,speed_ms,0,blend_radius_m)
    |   movel([0.254025, -1.225018, -2.665492, -0.821879, 1.570796, 1.824822],accel_mss,speed_ms,0,blend_radius_m)
    |   movel([0.255398, -1.224020, -2.665995, -0.822375, 1.570796, 1.826195],accel_mss,speed_ms,0,blend_radius_m)
    |   movel([0.256907, -1.223231, -2.666391, -0.822767, 1.570796, 1.827703],accel_mss,speed_ms,0,blend_radius_m)
    |   movel([0.258220, -1.222880, -2.666567, -0.822942, 1.570796, 1.829017],accel_mss,speed_ms,0,blend_radius_m)
    |   movel([0.259292, -1.222988, -2.666513, -0.822888, 1.570796, 1.830088],accel_mss,speed_ms,0,blend_radius_m)
    |   movel([0.260104, -1.223532, -2.666240, -0.822617, 1.570796, 1.830901],accel_mss,speed_ms,0,blend_radius_m)
    |   movel([0.260424, -1.223823, -2.666094, -0.822473, 1.570796, 1.831221],accel_mss,speed_ms,0,blend_radius_m)
    |   movel([0.260722, -1.223869, -2.666070, -0.822449, 1.570796, 1.831518],accel_mss,speed_ms,0,blend_radius_m)
    |   movel([0.261043, -1.223708, -2.666152, -0.822530, 1.570796, 1.831840],accel_mss,speed_ms,0,blend_radius_m)
    |   movel([0.261890, -1.222779, -2.666618, -0.822993, 1.570796, 1.832686],accel_mss,speed_ms,0,blend_radius_m)
    |   movel([0.262433, -1.223318, -2.666347, -0.822724, 1.570796, 1.833229],accel_mss,speed_ms,0,blend_radius_m)
    |   movel([0.262849, -1.223977, -2.666016, -0.822396, 1.570796, 1.833645],accel_mss,speed_ms,0,blend_radius_m)
    |   movel([0.263004, -1.224403, -2.665802, -0.822184, 1.570796, 1.833801],accel_mss,speed_ms,0,blend_radius_m)
    |   movel([0.263106, -1.225747, -2.665125, -0.821517, 1.570796, 1.833902],accel_mss,speed_ms,0,blend_radius_m)
    |   movel([0.262977, -1.227188, -2.664396, -0.820805, 1.570796, 1.833774],accel_mss,speed_ms,0,blend_radius_m)
    |   movel([0.262396, -1.230323, -2.662803, -0.819263, 1.570796, 1.833192],accel_mss,speed_ms,0,blend_radius_m)
    |   movel([0.262410, -1.230513, -2.662707, -0.819170, 1.570796, 1.833206],accel_mss,speed_ms,0,blend_radius_m)
    |   movel([0.262785, -1.230556, -2.662684, -0.819148, 1.570796, 1.833581],accel_mss,speed_ms,0,blend_radius_m)
    |   movel([0.263227, -1.230307, -2.662812, -0.819271, 1.570796, 1.834023],accel_mss,speed_ms,0,blend_radius_m)
    |   movel([0.263568, -1.229841, -2.663049, -0.819499, 1.570796, 1.834364],accel_mss,speed_ms,0,blend_radius_m)
    |   movel([0.263836, -1.229033, -2.663460, -0.819896, 1.570796, 1.834632],accel_mss,speed_ms,0,blend_radius_m)
    |   movel([0.264097, -1.227634, -2.664171, -0.820585, 1.570796, 1.834894],accel_mss,speed_ms,0,blend_radius_m)
    |   movel([0.264279, -1.226295, -2.664848, -0.821246, 1.570796, 1.835075],accel_mss,speed_ms,0,blend_radius_m)
    |   movel([0.264364, -1.224150, -2.665929, -0.822310, 1.570796, 1.835160],accel_mss,speed_ms,0,blend_radius_m)
    |   movel([0.264255, -1.223483, -2.666264, -0.822641, 1.570796, 1.835052],accel_mss,speed_ms,0,blend_radius_m)
    |   movel([0.263793, -1.222494, -2.666760, -0.823135, 1.570796, 1.834589],accel_mss,speed_ms,0,blend_radius_m)
    |   movel([0.263085, -1.221814, -2.667101, -0.823474, 1.570796, 1.833881],accel_mss,speed_ms,0,blend_radius_m)
    |   movel([0.262271, -1.221538, -2.667239, -0.823613, 1.570796, 1.833068],accel_mss,speed_ms,0,blend_radius_m)
    |   movel([0.261895, -1.221573, -2.667221, -0.823595, 1.570796, 1.832692],accel_mss,speed_ms,0,blend_radius_m)
    |   movel([0.261181, -1.221891, -2.667062, -0.823436, 1.570796, 1.831978],accel_mss,speed_ms,0,blend_radius_m)
    |   movel([0.260880, -1.221946, -2.667035, -0.823408, 1.570796, 1.831677],accel_mss,speed_ms,0,blend_radius_m)
    |   movel([0.260037, -1.221787, -2.667114, -0.823488, 1.570796, 1.830833],accel_mss,speed_ms,0,blend_radius_m)
    |   movel([0.259010, -1.221643, -2.667186, -0.823560, 1.570796, 1.829806],accel_mss,speed_ms,0,blend_radius_m)
    |   movel([0.257887, -1.221791, -2.667112, -0.823486, 1.570796, 1.828684],accel_mss,speed_ms,0,blend_radius_m)
    |   movel([0.256634, -1.222243, -2.666886, -0.823260, 1.570796, 1.827430],accel_mss,speed_ms,0,blend_radius_m)
    |   movel([0.253733, -1.223920, -2.666045, -0.822424, 1.570796, 1.824529],accel_mss,speed_ms,0,blend_radius_m)
    |   movel([0.252748, -1.220169, -2.667922, -0.824298, 1.570796, 1.823544],accel_mss,speed_ms,0,blend_radius_m)
    |   movel([0.251962, -1.216876, -2.669557, -0.825956, 1.570796, 1.822759],accel_mss,speed_ms,0,blend_radius_m)
    |   movel([0.251994, -1.216372, -2.669806, -0.826211, 1.570796, 1.822791],accel_mss,speed_ms,0,blend_radius_m)
    |   movel([0.252236, -1.216020, -2.669979, -0.826389, 1.570796, 1.823033],accel_mss,speed_ms,0,blend_radius_m)
    |   movel([0.252478, -1.215799, -2.670089, -0.826501, 1.570796, 1.823274],accel_mss,speed_ms,0,blend_radius_m)
    |   movel([0.252734, -1.215310, -2.670330, -0.826750, 1.570796, 1.823530],accel_mss,speed_ms,0,blend_radius_m)
    |   movel([0.252790, -1.214946, -2.670509, -0.826934, 1.570796, 1.823586],accel_mss,speed_ms,0,blend_radius_m)
    |   movel([0.253162, -1.213922, -2.671012, -0.827454, 1.570796, 1.823958],accel_mss,speed_ms,0,blend_radius_m)
    |   movel([0.253509, -1.213470, -2.671234, -0.827684, 1.570796, 1.824305],accel_mss,speed_ms,0,blend_radius_m)
    |   movel([0.253951, -1.213091, -2.671420, -0.827878, 1.570796, 1.824747],accel_mss,speed_ms,0,blend_radius_m)
    |   movel([0.254506, -1.212778, -2.671574, -0.828037, 1.570796, 1.825302],accel_mss,speed_ms,0,blend_radius_m)
    |   movel([0.255060, -1.212601, -2.671661, -0.828128, 1.570796, 1.825856],accel_mss,speed_ms,0,blend_radius_m)
    |   movel([0.256296, -1.212545, -2.671688, -0.828156, 1.570796, 1.827092],accel_mss,speed_ms,0,blend_radius_m)
    |   movel([0.257935, -1.212615, -2.671653, -0.828120, 1.570796, 1.828731],accel_mss,speed_ms,0,blend_radius_m)
    |   movel([0.258292, -1.212414, -2.671752, -0.828223, 1.570796, 1.829088],accel_mss,speed_ms,0,blend_radius_m)
    |   movel([0.258580, -1.212033, -2.671938, -0.828417, 1.570796, 1.829376],accel_mss,speed_ms,0,blend_radius_m)
    |   movel([0.259037, -1.211530, -2.672184, -0.828675, 1.570796, 1.829834],accel_mss,speed_ms,0,blend_radius_m)
    |   movel([0.259538, -1.211438, -2.672229, -0.828722, 1.570796, 1.830334],accel_mss,speed_ms,0,blend_radius_m)
    |   movel([0.260101, -1.211931, -2.671988, -0.828469, 1.570796, 1.830897],accel_mss,speed_ms,0,blend_radius_m)
    |   movel([0.260735, -1.213065, -2.671433, -0.827891, 1.570796, 1.831531],accel_mss,speed_ms,0,blend_radius_m)
    |   movel([0.261195, -1.214271, -2.670841, -0.827277, 1.570796, 1.831991],accel_mss,speed_ms,0,blend_radius_m)
    |   movel([0.261430, -1.215532, -2.670220, -0.826637, 1.570796, 1.832227],accel_mss,speed_ms,0,blend_radius_m)
    |   movel([0.261456, -1.216959, -2.669515, -0.825914, 1.570796, 1.832252],accel_mss,speed_ms,0,blend_radius_m)
    |   movel([0.261282, -1.218671, -2.668667, -0.825051, 1.570796, 1.832079],accel_mss,speed_ms,0,blend_radius_m)
    |   movel([0.261170, -1.219536, -2.668237, -0.824616, 1.570796, 1.831966],accel_mss,speed_ms,0,blend_radius_m)
    |   movel([0.261176, -1.220459, -2.667777, -0.824153, 1.570796, 1.831972],accel_mss,speed_ms,0,blend_radius_m)
    |   movel([0.261297, -1.220573, -2.667720, -0.824095, 1.570796, 1.832093],accel_mss,speed_ms,0,blend_radius_m)
    |   movel([0.261731, -1.220445, -2.667784, -0.824160, 1.570796, 1.832527],accel_mss,speed_ms,0,blend_radius_m)
    |   movel([0.262068, -1.220045, -2.667984, -0.824360, 1.570796, 1.832865],accel_mss,speed_ms,0,blend_radius_m)
    |   movel([0.262604, -1.218260, -2.668871, -0.825258, 1.570796, 1.833400],accel_mss,speed_ms,0,blend_radius_m)
    |   movel([0.262768, -1.215826, -2.670075, -0.826488, 1.570796, 1.833565],accel_mss,speed_ms,0,blend_radius_m)
    |   movel([0.262455, -1.213471, -2.671234, -0.827684, 1.570796, 1.833251],accel_mss,speed_ms,0,blend_radius_m)
    |   movel([0.262087, -1.212338, -2.671789, -0.828262, 1.570796, 1.832884],accel_mss,speed_ms,0,blend_radius_m)
    |   movel([0.261564, -1.211344, -2.672275, -0.828770, 1.570796, 1.832360],accel_mss,speed_ms,0,blend_radius_m)
    |   movel([0.260957, -1.210592, -2.672642, -0.829155, 1.570796, 1.831753],accel_mss,speed_ms,0,blend_radius_m)
    |   movel([0.260336, -1.210219, -2.672824, -0.829346, 1.570796, 1.831133],accel_mss,speed_ms,0,blend_radius_m)
    |   movel([0.259774, -1.210135, -2.672865, -0.829389, 1.570796, 1.830570],accel_mss,speed_ms,0,blend_radius_m)
    |   movel([0.259143, -1.210222, -2.672822, -0.829345, 1.570796, 1.829939],accel_mss,speed_ms,0,blend_radius_m)
    |   movel([0.258536, -1.210461, -2.672706, -0.829222, 1.570796, 1.829332],accel_mss,speed_ms,0,blend_radius_m)
    |   movel([0.257746, -1.211071, -2.672409, -0.828910, 1.570796, 1.828542],accel_mss,speed_ms,0,blend_radius_m)
    |   movel([0.257492, -1.211199, -2.672346, -0.828844, 1.570796, 1.828288],accel_mss,speed_ms,0,blend_radius_m)
    |   movel([0.256565, -1.211239, -2.672326, -0.828824, 1.570796, 1.827361],accel_mss,speed_ms,0,blend_radius_m)
    |   movel([0.256098, -1.211245, -2.672324, -0.828821, 1.570796, 1.826894],accel_mss,speed_ms,0,blend_radius_m)
    |   movel([0.254741, -1.211528, -2.672185, -0.828676, 1.570796, 1.825538],accel_mss,speed_ms,0,blend_radius_m)
    |   movel([0.253907, -1.211979, -2.671965, -0.828445, 1.570796, 1.824703],accel_mss,speed_ms,0,blend_radius_m)
    |   movel([0.253034, -1.212673, -2.671625, -0.828091, 1.570796, 1.823830],accel_mss,speed_ms,0,blend_radius_m)
    |   movel([0.252279, -1.213473, -2.671233, -0.827683, 1.570796, 1.823075],accel_mss,speed_ms,0,blend_radius_m)
    |   movel([0.251415, -1.215030, -2.670467, -0.826891, 1.570796, 1.822212],accel_mss,speed_ms,0,blend_radius_m)
    |   movel([0.250557, -1.212719, -2.671603, -0.828068, 1.570796, 1.821354],accel_mss,speed_ms,0,blend_radius_m)
    |   movel([0.248798, -1.208537, -2.673641, -0.830211, 1.570796, 1.819595],accel_mss,speed_ms,0,blend_radius_m)
    |   movel([0.248201, -1.207161, -2.674308, -0.830920, 1.570796, 1.818997],accel_mss,speed_ms,0,blend_radius_m)
    |   movel([0.248062, -1.206328, -2.674710, -0.831351, 1.570796, 1.818858],accel_mss,speed_ms,0,blend_radius_m)
    |   movel([0.248283, -1.205665, -2.675030, -0.831694, 1.570796, 1.819079],accel_mss,speed_ms,0,blend_radius_m)
    |   movel([0.248858, -1.204999, -2.675351, -0.832039, 1.570796, 1.819654],accel_mss,speed_ms,0,blend_radius_m)
    |   movel([0.249571, -1.204524, -2.675579, -0.832285, 1.570796, 1.820367],accel_mss,speed_ms,0,blend_radius_m)
    |   movel([0.250384, -1.204224, -2.675724, -0.832441, 1.570796, 1.821181],accel_mss,speed_ms,0,blend_radius_m)
    |   movel([0.251262, -1.204111, -2.675778, -0.832500, 1.570796, 1.822059],accel_mss,speed_ms,0,blend_radius_m)
    |   movel([0.252158, -1.204197, -2.675737, -0.832456, 1.570796, 1.822955],accel_mss,speed_ms,0,blend_radius_m)
    |   movel([0.252933, -1.204296, -2.675689, -0.832404, 1.570796, 1.823729],accel_mss,speed_ms,0,blend_radius_m)
    |   movel([0.253423, -1.204171, -2.675749, -0.832469, 1.570796, 1.824219],accel_mss,speed_ms,0,blend_radius_m)
    |   movel([0.253763, -1.203839, -2.675909, -0.832642, 1.570796, 1.824559],accel_mss,speed_ms,0,blend_radius_m)
    |   movel([0.254337, -1.202442, -2.676578, -0.833369, 1.570796, 1.825134],accel_mss,speed_ms,0,blend_radius_m)
    |   movel([0.254877, -1.202185, -2.676701, -0.833503, 1.570796, 1.825674],accel_mss,speed_ms,0,blend_radius_m)
    |   movel([0.255669, -1.202383, -2.676606, -0.833400, 1.570796, 1.826465],accel_mss,speed_ms,0,blend_radius_m)
    |   movel([0.257172, -1.203231, -2.676200, -0.832958, 1.570796, 1.827969],accel_mss,speed_ms,0,blend_radius_m)
    |   movel([0.257876, -1.204066, -2.675799, -0.832523, 1.570796, 1.828673],accel_mss,speed_ms,0,blend_radius_m)
    |   movel([0.258228, -1.204977, -2.675362, -0.832051, 1.570796, 1.829025],accel_mss,speed_ms,0,blend_radius_m)
    |   movel([0.258271, -1.206129, -2.674806, -0.831453, 1.570796, 1.829067],accel_mss,speed_ms,0,blend_radius_m)
    |   movel([0.257734, -1.209382, -2.673231, -0.829776, 1.570796, 1.828530],accel_mss,speed_ms,0,blend_radius_m)
    |   movel([0.257825, -1.209583, -2.673133, -0.829672, 1.570796, 1.828621],accel_mss,speed_ms,0,blend_radius_m)
    |   movel([0.258055, -1.209639, -2.673106, -0.829644, 1.570796, 1.828852],accel_mss,speed_ms,0,blend_radius_m)
    |   movel([0.258461, -1.209436, -2.673205, -0.829748, 1.570796, 1.829257],accel_mss,speed_ms,0,blend_radius_m)
    |   movel([0.258801, -1.208989, -2.673422, -0.829978, 1.570796, 1.829597],accel_mss,speed_ms,0,blend_radius_m)
    |   movel([0.259103, -1.208186, -2.673812, -0.830391, 1.570796, 1.829899],accel_mss,speed_ms,0,blend_radius_m)
    |   movel([0.259567, -1.206002, -2.674868, -0.831519, 1.570796, 1.830364],accel_mss,speed_ms,0,blend_radius_m)
    |   movel([0.259625, -1.205325, -2.675194, -0.831870, 1.570796, 1.830422],accel_mss,speed_ms,0,blend_radius_m)
    |   movel([0.259490, -1.204093, -2.675787, -0.832510, 1.570796, 1.830287],accel_mss,speed_ms,0,blend_radius_m)
    |   movel([0.258855, -1.202668, -2.676469, -0.833251, 1.570796, 1.829651],accel_mss,speed_ms,0,blend_radius_m)
    |   movel([0.257727, -1.201598, -2.676981, -0.833810, 1.570796, 1.828523],accel_mss,speed_ms,0,blend_radius_m)
    |   movel([0.256299, -1.201020, -2.677257, -0.834112, 1.570796, 1.827095],accel_mss,speed_ms,0,blend_radius_m)
    |   movel([0.255578, -1.200958, -2.677287, -0.834144, 1.570796, 1.826374],accel_mss,speed_ms,0,blend_radius_m)
    |   movel([0.254778, -1.201063, -2.677236, -0.834089, 1.570796, 1.825575],accel_mss,speed_ms,0,blend_radius_m)
    |   movel([0.253898, -1.201362, -2.677094, -0.833933, 1.570796, 1.824694],accel_mss,speed_ms,0,blend_radius_m)
    |   movel([0.253681, -1.201588, -2.676986, -0.833815, 1.570796, 1.824477],accel_mss,speed_ms,0,blend_radius_m)
    |   movel([0.253182, -1.202462, -2.676568, -0.833359, 1.570796, 1.823978],accel_mss,speed_ms,0,blend_radius_m)
    |   movel([0.253004, -1.202670, -2.676469, -0.833250, 1.570796, 1.823800],accel_mss,speed_ms,0,blend_radius_m)
    |   movel([0.252516, -1.202803, -2.676405, -0.833181, 1.570796, 1.823313],accel_mss,speed_ms,0,blend_radius_m)
    |   movel([0.251099, -1.202890, -2.676363, -0.833136, 1.570796, 1.821895],accel_mss,speed_ms,0,blend_radius_m)
    |   movel([0.250048, -1.203155, -2.676237, -0.832998, 1.570796, 1.820845],accel_mss,speed_ms,0,blend_radius_m)
    |   movel([0.249115, -1.203652, -2.675998, -0.832739, 1.570796, 1.819912],accel_mss,speed_ms,0,blend_radius_m)
    |   movel([0.248109, -1.204462, -2.675609, -0.832318, 1.570796, 1.818905],accel_mss,speed_ms,0,blend_radius_m)
    |   movel([0.247125, -1.205374, -2.675171, -0.831845, 1.570796, 1.817921],accel_mss,speed_ms,0,blend_radius_m)
    |   movel([0.245954, -1.203671, -2.675989, -0.832729, 1.570796, 1.816750],accel_mss,speed_ms,0,blend_radius_m)
    |   movel([0.244479, -1.201769, -2.676900, -0.833721, 1.570796, 1.815275],accel_mss,speed_ms,0,blend_radius_m)
    |   movel([0.240414, -1.197694, -2.678837, -0.835858, 1.570796, 1.811210],accel_mss,speed_ms,0,blend_radius_m)
    |   movel([0.238447, -1.196147, -2.679568, -0.836674, 1.570796, 1.809243],accel_mss,speed_ms,0,blend_radius_m)
    |   movel([0.234488, -1.193797, -2.680673, -0.837920, 1.570796, 1.805284],accel_mss,speed_ms,0,blend_radius_m)
    |   movel([0.229979, -1.191909, -2.681556, -0.838924, 1.570796, 1.800775],accel_mss,speed_ms,0,blend_radius_m)
    |   movel([0.224976, -1.190532, -2.682198, -0.839659, 1.570796, 1.795772],accel_mss,speed_ms,0,blend_radius_m)
    |   movel([0.219555, -1.189684, -2.682592, -0.840113, 1.570796, 1.790351],accel_mss,speed_ms,0,blend_radius_m)
    |   movel([0.217106, -1.189333, -2.682755, -0.840301, 1.570796, 1.787902],accel_mss,speed_ms,0,blend_radius_m)
    |   movel([0.217224, -1.187364, -2.683667, -0.841358, 1.570796, 1.788021],accel_mss,speed_ms,0,blend_radius_m)
    |   movel([0.217387, -1.186835, -2.683911, -0.841643, 1.570796, 1.788183],accel_mss,speed_ms,0,blend_radius_m)
    |   movel([0.218140, -1.185484, -2.684534, -0.842372, 1.570796, 1.788937],accel_mss,speed_ms,0,blend_radius_m)
    |   movel([0.218922, -1.184422, -2.685021, -0.842946, 1.570796, 1.789718],accel_mss,speed_ms,0,blend_radius_m)
    |   movel([0.219878, -1.183424, -2.685479, -0.843486, 1.570796, 1.790674],accel_mss,speed_ms,0,blend_radius_m)
    |   movel([0.220918, -1.182581, -2.685864, -0.843944, 1.570796, 1.791715],accel_mss,speed_ms,0,blend_radius_m)
    |   movel([0.221947, -1.181971, -2.686143, -0.844276, 1.570796, 1.792744],accel_mss,speed_ms,0,blend_radius_m)
    |   movel([0.222470, -1.181650, -2.686289, -0.844450, 1.570796, 1.793266],accel_mss,speed_ms,0,blend_radius_m)
    |   movel([0.222774, -1.181299, -2.686449, -0.844641, 1.570796, 1.793570],accel_mss,speed_ms,0,blend_radius_m)
    |   movel([0.222894, -1.180866, -2.686646, -0.844877, 1.570796, 1.793690],accel_mss,speed_ms,0,blend_radius_m)
    |   movel([0.222829, -1.180295, -2.686906, -0.845188, 1.570796, 1.793625],accel_mss,speed_ms,0,blend_radius_m)
    |   movel([0.222886, -1.179314, -2.687351, -0.845724, 1.570796, 1.793683],accel_mss,speed_ms,0,blend_radius_m)
    |   movel([0.223406, -1.178170, -2.687869, -0.846350, 1.570796, 1.794202],accel_mss,speed_ms,0,blend_radius_m)
    |   movel([0.224330, -1.177003, -2.688396, -0.846990, 1.570796, 1.795126],accel_mss,speed_ms,0,blend_radius_m)
    |   movel([0.225545, -1.175966, -2.688863, -0.847560, 1.570796, 1.796342],accel_mss,speed_ms,0,blend_radius_m)
    |   movel([0.225846, -1.175788, -2.688943, -0.847658, 1.570796, 1.796642],accel_mss,speed_ms,0,blend_radius_m)
    |   movel([0.227519, -1.175169, -2.689221, -0.847999, 1.570796, 1.798315],accel_mss,speed_ms,0,blend_radius_m)
    |   movel([0.228859, -1.174940, -2.689324, -0.848125, 1.570796, 1.799656],accel_mss,speed_ms,0,blend_radius_m)
    |   movel([0.230085, -1.175038, -2.689280, -0.848071, 1.570796, 1.800881],accel_mss,speed_ms,0,blend_radius_m)
